u16gPvgArrowArmVoltage.AppScalingDivisor :=1;
u16gPvgArrowArmVoltage.AppScalingMultiplier :=1;
u16gPvgArrowArmVoltage.AppScalingOffset :=0;
u16gPvgArrowArmVoltage.AppUnit :="";
u16gPvgArrowArmVoltage.CanDefault :=0;
u16gPvgArrowArmVoltage.CanInit :=0;
u16gPvgArrowArmVoltage.CanMax :=VBasic.LibConst.U16_MAX;
u16gPvgArrowArmVoltage.CanMin :=VBasic.LibConst.U16_MIN;
u16gPvgArrowArmVoltage.CanUnit :="";
u16gPvgArrowArmVoltage.Description :="new signal";
u16gPvgArrowArmVoltage.ErrorReaction := eErrorReaction.ERSIG_DFLT;
u16gPvgArrowArmVoltage.ReceiverAdress :=1;
u16gPvgArrowArmVoltage.ToolScalingDivisor :=1;
u16gPvgArrowArmVoltage.ToolScalingMultiplier :=1;
u16gPvgArrowArmVoltage.ToolScalingOffset :=0;
u16gPvgArrowArmVoltage.ToolUnit :="";

u16gPvgTelescopeArmVoltage.AppScalingDivisor :=1;
u16gPvgTelescopeArmVoltage.AppScalingMultiplier :=1;
u16gPvgTelescopeArmVoltage.AppScalingOffset :=0;
u16gPvgTelescopeArmVoltage.AppUnit :="";
u16gPvgTelescopeArmVoltage.CanDefault :=0;
u16gPvgTelescopeArmVoltage.CanInit :=0;
u16gPvgTelescopeArmVoltage.CanMax :=VBasic.LibConst.U16_MAX;
u16gPvgTelescopeArmVoltage.CanMin :=VBasic.LibConst.U16_MIN;
u16gPvgTelescopeArmVoltage.CanUnit :="";
u16gPvgTelescopeArmVoltage.Description :="new signal";
u16gPvgTelescopeArmVoltage.ErrorReaction := eErrorReaction.ERSIG_DFLT;
u16gPvgTelescopeArmVoltage.ReceiverAdress :=1;
u16gPvgTelescopeArmVoltage.ToolScalingDivisor :=1;
u16gPvgTelescopeArmVoltage.ToolScalingMultiplier :=1;
u16gPvgTelescopeArmVoltage.ToolScalingOffset :=0;
u16gPvgTelescopeArmVoltage.ToolUnit :="";

u16gPvgEvTorVoltage.AppScalingDivisor :=1;
u16gPvgEvTorVoltage.AppScalingMultiplier :=1;
u16gPvgEvTorVoltage.AppScalingOffset :=0;
u16gPvgEvTorVoltage.AppUnit :="";
u16gPvgEvTorVoltage.CanDefault :=0;
u16gPvgEvTorVoltage.CanInit :=0;
u16gPvgEvTorVoltage.CanMax :=VBasic.LibConst.U16_MAX;
u16gPvgEvTorVoltage.CanMin :=VBasic.LibConst.U16_MIN;
u16gPvgEvTorVoltage.CanUnit :="";
u16gPvgEvTorVoltage.Description :="new signal";
u16gPvgEvTorVoltage.ErrorReaction := eErrorReaction.ERSIG_DFLT;
u16gPvgEvTorVoltage.ReceiverAdress :=1;
u16gPvgEvTorVoltage.ToolScalingDivisor :=1;
u16gPvgEvTorVoltage.ToolScalingMultiplier :=1;
u16gPvgEvTorVoltage.ToolScalingOffset :=0;
u16gPvgEvTorVoltage.ToolUnit :="";


                
END_METHOD
END_FUNCTION_BLOCK

FUNCTION_BLOCK Msg9C1SendToEvision7MessageClass EXTENDS CanReceiveMessageClass
  VAR_INPUT
    bogPendularMoveUp : BoolCanSignalClass;
    bogPendularMoveDown : BoolCanSignalClass;
    bogBasketRotCtClockWiseMove : BoolCanSignalClass;
    bogBasketRtClockWiseMove : BoolCanSignalClass;
    bogBasketInclinaisonMoveUp : BoolCanSignalClass;
    bogBasketInclinaisonMoveDown : BoolCanSignalClass;
    bogFuelLow : BoolCanSignalClass;
    i16gDeltaArmAngleValue : Int16CanSignalClass;
    i16gArrowArmAngleValue : Int16CanSignalClass;
    i16gTelescopePositionValue : Int16CanSignalClass;
    Counter : UInt32CanSignalClass;
  END_VAR

            
          

METHOD SetData
  VAR_INPUT
    CanMsgPointer : POINTER TO CanMessageClass;
  END_VAR
                  IF IsValidPointer(canMsgPointer,'SetData') THEN
	SUPER^.SetData(CanMsgPointer);
	//Set the new data
	bogPendularMoveUp.Value := canMsgPointer^.GetBoolOnBit(0);
	bogPendularMoveDown.Value := canMsgPointer^.GetBoolOnBit(1);
	bogBasketRotCtClockWiseMove.Value := canMsgPointer^.GetBoolOnBit(2);
	bogBasketRtClockWiseMove.Value := canMsgPointer^.GetBoolOnBit(3);
	bogBasketInclinaisonMoveUp.Value := canMsgPointer^.GetBoolOnBit(4);
	bogBasketInclinaisonMoveDown.Value := canMsgPointer^.GetBoolOnBit(5);
	bogFuelLow.Value := canMsgPointer^.GetBoolOnBit(6);
	i16gDeltaArmAngleValue.Value := canMsgPointer^.GetInt16(16);
	i16gArrowArmAngleValue.Value := canMsgPointer^.GetInt16(32);
	i16gTelescopePositionValue.Value := canMsgPointer^.GetInt16(48);
	//And increase the counter
	Counter.Value := CanMsgPointer^.Counter.Value;
END_IF

                
END_METHOD

PROPERTY bogPendularMoveUpRawValue : BOOL
GET
                    bogPendularMoveUpRawValue := bogPendularMoveUp.Value;

                  
END_GET
END_PROPERTY

PROPERTY bogPendularMoveDownRawValue : BOOL
GET
                    bogPendularMoveDownRawValue := bogPendularMoveDown.Value;

                  
END_GET
END_PROPERTY

PROPERTY bogBasketRotCtClockWiseMoveRawValue : BOOL
GET
                    bogBasketRotCtClockWiseMoveRawValue := bogBasketRotCtClockWiseMove.Value;

                  
END_GET
END_PROPERTY

PROPERTY bogBasketRtClockWiseMoveRawValue : BOOL
GET
                    bogBasketRtClockWiseMoveRawValue := bogBasketRtClockWiseMove.Value;

                  
END_GET
END_PROPERTY

PROPERTY bogBasketInclinaisonMoveUpRawValue : BOOL
GET
                    bogBasketInclinaisonMoveUpRawValue := bogBasketInclinaisonMoveUp.Value;

                  
END_GET
END_PROPERTY

PROPERTY bogBasketInclinaisonMoveDownRawValue : BOOL
GET
                    bogBasketInclinaisonMoveDownRawValue := bogBasketInclinaisonMoveDown.Value;

                  
END_GET
END_PROPERTY

PROPERTY bogFuelLowRawValue : BOOL
GET
                    bogFuelLowRawValue := bogFuelLow.Value;

                  
END_GET
END_PROPERTY

PROPERTY i16gDeltaArmAngleValueRawValue : INT
GET
                    IF i16gDeltaArmAngleValue.AppScalingMultiplier = 0 THEN
	_MatchLog^.Error("Get i16gDeltaArmAngleValueRawValue", "Division by Zero!");
	RETURN;
End_IF

i16gDeltaArmAngleValueRawValue := TO_INT((i16gDeltaArmAngleValue.Value - i16gDeltaArmAngleValue.AppScalingOffset) * i16gDeltaArmAngleValue.AppScalingDivisor / i16gDeltaArmAngleValue.AppScalingMultiplier);

                  
END_GET
END_PROPERTY

PROPERTY i16gArrowArmAngleValueRawValue : INT
GET
                    IF i16gArrowArmAngleValue.AppScalingMultiplier = 0 THEN
	_MatchLog^.Error("Get i16gArrowArmAngleValueRawValue", "Division by Zero!");
	RETURN;
End_IF

i16gArrowArmAngleValueRawValue := TO_INT((i16gArrowArmAngleValue.Value - i16gArrowArmAngleValue.AppScalingOffset) * i16gArrowArmAngleValue.AppScalingDivisor / i16gArrowArmAngleValue.AppScalingMultiplier);

                  
END_GET
END_PROPERTY

PROPERTY i16gTelescopePositionValueRawValue : INT
GET
                    IF i16gTelescopePositionValue.AppScalingMultiplier = 0 THEN
	_MatchLog^.Error("Get i16gTelescopePositionValueRawValue", "Division by Zero!");
	RETURN;
End_IF

i16gTelescopePositionValueRawValue := TO_INT((i16gTelescopePositionValue.Value - i16gTelescopePositionValue.AppScalingOffset) * i16gTelescopePositionValue.AppScalingDivisor / i16gTelescopePositionValue.AppScalingMultiplier);

                  
END_GET
END_PROPERTY

PROPERTY bogPendularMoveUpToolValue : BOOL
GET
                    bogPendularMoveUpToolValue := bogPendularMoveUp.Value;

                  
END_GET
END_PROPERTY

PROPERTY bogPendularMoveDownToolValue : BOOL
GET
                    bogPendularMoveDownToolValue := bogPendularMoveDown.Value;

                  
END_GET
END_PROPERTY

PROPERTY bogBasketRotCtClockWiseMoveToolValue : BOOL
GET
                    bogBasketRotCtClockWiseMoveToolValue := bogBasketRotCtClockWiseMove.Value;

                  
END_GET
END_PROPERTY

PROPERTY bogBasketRtClockWiseMoveToolValue : BOOL
GET
                    bogBasketRtClockWiseMoveToolValue := bogBasketRtClockWiseMove.Value;

                  
END_GET
END_PROPERTY

PROPERTY bogBasketInclinaisonMoveUpToolValue : BOOL
GET
                    bogBasketInclinaisonMoveUpToolValue := bogBasketInclinaisonMoveUp.Value;

                  
END_GET
END_PROPERTY

PROPERTY bogBasketInclinaisonMoveDownToolValue : BOOL
GET
                    bogBasketInclinaisonMoveDownToolValue := bogBasketInclinaisonMoveDown.Value;

                  
END_GET
END_PROPERTY

PROPERTY bogFuelLowToolValue : BOOL
GET
                    bogFuelLowToolValue := bogFuelLow.Value;

                  
END_GET
END_PROPERTY

PROPERTY i16gDeltaArmAngleValueToolValue : INT
GET
                    IF i16gDeltaArmAngleValue.ToolScalingDivisor = 0 OR i16gDeltaArmAngleValue.AppScalingMultiplier = 0 THEN
	_MatchLog^.Error("Get i16gDeltaArmAngleValueToolValue", "Division by Zero!");
	RETURN;
END_IF

i16gDeltaArmAngleValueToolValue := TO_INT(((i16gDeltaArmAngleValue.Value - i16gDeltaArmAngleValue.AppScalingOffset) * i16gDeltaArmAngleValue.AppScalingDivisor / i16gDeltaArmAngleValue.AppScalingMultiplier * i16gDeltaArmAngleValue.ToolScalingMultiplier / i16gDeltaArmAngleValue.ToolScalingDivisor) + i16gDeltaArmAngleValue.ToolScalingOffset);

                  
END_GET
END_PROPERTY

PROPERTY i16gArrowArmAngleValueToolValue : INT
GET
                    IF i16gArrowArmAngleValue.ToolScalingDivisor = 0 OR i16gArrowArmAngleValue.AppScalingMultiplier = 0 THEN
	_MatchLog^.Error("Get i16gArrowArmAngleValueToolValue", "Division by Zero!");
	RETURN;
END_IF

i16gArrowArmAngleValueToolValue := TO_INT(((i16gArrowArmAngleValue.Value - i16gArrowArmAngleValue.AppScalingOffset) * i16gArrowArmAngleValue.AppScalingDivisor / i16gArrowArmAngleValue.AppScalingMultiplier * i16gArrowArmAngleValue.ToolScalingMultiplier / i16gArrowArmAngleValue.ToolScalingDivisor) + i16gArrowArmAngleValue.ToolScalingOffset);

                  
END_GET
END_PROPERTY

PROPERTY i16gTelescopePositionValueToolValue : INT
GET
                    IF i16gTelescopePositionValue.ToolScalingDivisor = 0 OR i16gTelescopePositionValue.AppScalingMultiplier = 0 THEN
	_MatchLog^.Error("Get i16gTelescopePositionValueToolValue", "Division by Zero!");
	RETURN;
END_IF

i16gTelescopePositionValueToolValue := TO_INT(((i16gTelescopePositionValue.Value - i16gTelescopePositionValue.AppScalingOffset) * i16gTelescopePositionValue.AppScalingDivisor / i16gTelescopePositionValue.AppScalingMultiplier * i16gTelescopePositionValue.ToolScalingMultiplier / i16gTelescopePositionValue.ToolScalingDivisor) + i16gTelescopePositionValue.ToolScalingOffset);

                  
END_GET
END_PROPERTY

METHOD InitializeCanSignals
                  bogPendularMoveUp.AppScalingDivisor :=1;
bogPendularMoveUp.AppScalingMultiplier :=1;
bogPendularMoveUp.AppScalingOffset :=0;
bogPendularMoveUp.AppUnit :="";
bogPendularMoveUp.CanDefault :=0;
bogPendularMoveUp.CanInit :=0;
bogPendularMoveUp.CanMax :=1;
bogPendularMoveUp.CanMin :=0;
bogPendularMoveUp.CanUnit :="";
bogPendularMoveUp.Description :="new signal";
bogPendularMoveUp.ErrorReaction := eErrorReaction.ERSIG_DFLT;
bogPendularMoveUp.ReceiverAdress :=1;
bogPendularMoveUp.ToolScalingDivisor :=1;
bogPendularMoveUp.ToolScalingMultiplier :=1;
bogPendularMoveUp.ToolScalingOffset :=0;
bogPendularMoveUp.ToolUnit :="";

bogPendularMoveDown.AppScalingDivisor :=1;
bogPendularMoveDown.AppScalingMultiplier :=1;
bogPendularMoveDown.AppScalingOffset :=0;
bogPendularMoveDown.AppUnit :="";
bogPendularMoveDown.CanDefault :=0;
bogPendularMoveDown.CanInit :=0;
bogPendularMoveDown.CanMax :=1;
bogPendularMoveDown.CanMin :=0;
bogPendularMoveDown.CanUnit :="";
bogPendularMoveDown.Description :="new signal";
bogPendularMoveDown.ErrorReaction := eErrorReaction.ERSIG_DFLT;
bogPendularMoveDown.ReceiverAdress :=1;
bogPendularMoveDown.ToolScalingDivisor :=1;
bogPendularMoveDown.ToolScalingMultiplier :=1;
bogPendularMoveDown.ToolScalingOffset :=0;
bogPendularMoveDown.ToolUnit :="";

bogBasketRotCtClockWiseMove.AppScalingDivisor :=1;
bogBasketRotCtClockWiseMove.AppScalingMultiplier :=1;
bogBasketRotCtClockWiseMove.AppScalingOffset :=0;
bogBasketRotCtClockWiseMove.AppUnit :="";
bogBasketRotCtClockWiseMove.CanDefault :=0;
bogBasketRotCtClockWiseMove.CanInit :=0;
bogBasketRotCtClockWiseMove.CanMax :=1;
bogBasketRotCtClockWiseMove.CanMin :=0;
bogBasketRotCtClockWiseMove.CanUnit :="";
bogBasketRotCtClockWiseMove.Description :="new signal";
bogBasketRotCtClockWiseMove.ErrorReaction := eErrorReaction.ERSIG_DFLT;
bogBasketRotCtClockWiseMove.ReceiverAdress :=1;
bogBasketRotCtClockWiseMove.ToolScalingDivisor :=1;
bogBasketRotCtClockWiseMove.ToolScalingMultiplier :=1;
bogBasketRotCtClockWiseMove.ToolScalingOffset :=0;
bogBasketRotCtClockWiseMove.ToolUnit :="";

bogBasketRtClockWiseMove.AppScalingDivisor :=1;
bogBasketRtClockWiseMove.AppScalingMultiplier :=1;
bogBasketRtClockWiseMove.AppScalingOffset :=0;
bogBasketRtClockWiseMove.AppUnit :="";
bogBasketRtClockWiseMove.CanDefault :=0;
bogBasketRtClockWiseMove.CanInit :=0;
bogBasketRtClockWiseMove.CanMax :=1;
bogBasketRtClockWiseMove.CanMin :=0;
bogBasketRtClockWiseMove.CanUnit :="";
bogBasketRtClockWiseMove.Description :="new signal";
bogBasketRtClockWiseMove.ErrorReaction := eErrorReaction.ERSIG_DFLT;
bogBasketRtClockWiseMove.ReceiverAdress :=1;
bogBasketRtClockWiseMove.ToolScalingDivisor :=1;
bogBasketRtClockWiseMove.ToolScalingMultiplier :=1;
bogBasketRtClockWiseMove.ToolScalingOffset :=0;
bogBasketRtClockWiseMove.ToolUnit :="";

bogBasketInclinaisonMoveUp.AppScalingDivisor :=1;
bogBasketInclinaisonMoveUp.AppScalingMultiplier :=1;
bogBasketInclinaisonMoveUp.AppScalingOffset :=0;
bogBasketInclinaisonMoveUp.AppUnit :="";
bogBasketInclinaisonMoveUp.CanDefault :=0;
bogBasketInclinaisonMoveUp.CanInit :=0;
bogBasketInclinaisonMoveUp.CanMax :=1;
bogBasketInclinaisonMoveUp.CanMin :=0;
bogBasketInclinaisonMoveUp.CanUnit :="";
bogBasketInclinaisonMoveUp.Description :="new signal";
bogBasketInclinaisonMoveUp.ErrorReaction := eErrorReaction.ERSIG_DFLT;
bogBasketInclinaisonMoveUp.ReceiverAdress :=1;
bogBasketInclinaisonMoveUp.ToolScalingDivisor :=1;
bogBasketInclinaisonMoveUp.ToolScalingMultiplier :=1;
bogBasketInclinaisonMoveUp.ToolScalingOffset :=0;
bogBasketInclinaisonMoveUp.ToolUnit :="";

bogBasketInclinaisonMoveDown.AppScalingDivisor :=1;
bogBasketInclinaisonMoveDown.AppScalingMultiplier :=1;
bogBasketInclinaisonMoveDown.AppScalingOffset :=0;
bogBasketInclinaisonMoveDown.AppUnit :="";
bogBasketInclinaisonMoveDown.CanDefault :=0;
bogBasketInclinaisonMoveDown.CanInit :=0;
bogBasketInclinaisonMoveDown.CanMax :=1;
bogBasketInclinaisonMoveDown.CanMin :=0;
bogBasketInclinaisonMoveDown.CanUnit :="";
bogBasketInclinaisonMoveDown.Description :="new signal";
bogBasketInclinaisonMoveDown.ErrorReaction := eErrorReaction.ERSIG_DFLT;
bogBasketInclinaisonMoveDown.ReceiverAdress :=1;
bogBasketInclinaisonMoveDown.ToolScalingDivisor :=1;
bogBasketInclinaisonMoveDown.ToolScalingMultiplier :=1;
bogBasketInclinaisonMoveDown.ToolScalingOffset :=0;
bogBasketInclinaisonMoveDown.ToolUnit :="";

bogFuelLow.AppScalingDivisor :=1;
bogFuelLow.AppScalingMultiplier :=1;
bogFuelLow.AppScalingOffset :=0;
bogFuelLow.AppUnit :="";
bogFuelLow.CanDefault :=0;
bogFuelLow.CanInit :=0;
bogFuelLow.CanMax :=1;
bogFuelLow.CanMin :=0;
bogFuelLow.CanUnit :="";
bogFuelLow.Description :="new signal";
bogFuelLow.ErrorReaction := eErrorReaction.ERSIG_DFLT;
bogFuelLow.ReceiverAdress :=1;
bogFuelLow.ToolScalingDivisor :=1;
bogFuelLow.ToolScalingMultiplier :=1;
bogFuelLow.ToolScalingOffset :=0;
bogFuelLow.ToolUnit :="";

i16gDeltaArmAngleValue.AppScalingDivisor :=1;
i16gDeltaArmAngleValue.AppScalingMultiplier :=1;
i16gDeltaArmAngleValue.AppScalingOffset :=0;
i16gDeltaArmAngleValue.AppUnit :="";
i16gDeltaArmAngleValue.CanDefault :=0;
i16gDeltaArmAngleValue.CanInit :=0;
i16gDeltaArmAngleValue.CanMax :=VBasic.LibConst.I16_MAX;
i16gDeltaArmAngleValue.CanMin :=VBasic.LibConst.I16_MIN;
i16gDeltaArmAngleValue.CanUnit :="";
i16gDeltaArmAngleValue.Description :="new signal";
i16gDeltaArmAngleValue.ErrorReaction := eErrorReaction.ERSIG_DFLT;
i16gDeltaArmAngleValue.ReceiverAdress :=1;
i16gDeltaArmAngleValue.ToolScalingDivisor :=1;
i16gDeltaArmAngleValue.ToolScalingMultiplier :=1;
i16gDeltaArmAngleValue.ToolScalingOffset :=0;
i16gDeltaArmAngleValue.ToolUnit :="";

i16gArrowArmAngleValue.AppScalingDivisor :=1;
i16gArrowArmAngleValue.AppScalingMultiplier :=1;
i16gArrowArmAngleValue.AppScalingOffset :=0;
i16gArrowArmAngleValue.AppUnit :="";
i16gArrowArmAngleValue.CanDefault :=0;
i16gArrowArmAngleValue.CanInit :=0;
i16gArrowArmAngleValue.CanMax :=VBasic.LibConst.I16_MAX;
i16gArrowArmAngleValue.CanMin :=VBasic.LibConst.I16_MIN;
i16gArrowArmAngleValue.CanUnit :="";
i16gArrowArmAngleValue.Description :="new signal";
i16gArrowArmAngleValue.ErrorReaction := eErrorReaction.ERSIG_DFLT;
i16gArrowArmAngleValue.ReceiverAdress :=1;
i16gArrowArmAngleValue.ToolScalingDivisor :=1;
i16gArrowArmAngleValue.ToolScalingMultiplier :=1;
i16gArrowArmAngleValue.ToolScalingOffset :=0;
i16gArrowArmAngleValue.ToolUnit :="";

i16gTelescopePositionValue.AppScalingDivisor :=1;
i16gTelescopePositionValue.AppScalingMultiplier :=1;
i16gTelescopePositionValue.AppScalingOffset :=0;
i16gTelescopePositionValue.AppUnit :="";
i16gTelescopePositionValue.CanDefault :=0;
i16gTelescopePositionValue.CanInit :=0;
i16gTelescopePositionValue.CanMax :=VBasic.LibConst.I16_MAX;
i16gTelescopePositionValue.CanMin :=VBasic.LibConst.I16_MIN;
i16gTelescopePositionValue.CanUnit :="";
i16gTelescopePositionValue.Description :="new signal";
i16gTelescopePositionValue.ErrorReaction := eErrorReaction.ERSIG_DFLT;
i16gTelescopePositionValue.ReceiverAdress :=1;
i16gTelescopePositionValue.ToolScalingDivisor :=1;
i16gTelescopePositionValue.ToolScalingMultiplier :=1;
i16gTelescopePositionValue.ToolScalingOffset :=0;
i16gTelescopePositionValue.ToolUnit :="";


                
END_METHOD
END_FUNCTION_BLOCK

FUNCTION_BLOCK Msg10C1SendToEvision7MessageClass EXTENDS CanReceiveMessageClass
  VAR_INPUT
    u8gTTC510Version_Major : UInt8CanSignalClass;
    u8gTTC510Version_Minor : UInt8CanSignalClass;
    u8gTTC510Version_Patch : UInt8CanSignalClass;
    u8gTTC510Version_Custom : UInt8CanSignalClass;
    u8gTTC48XSVersion_Major : UInt8CanSignalClass;
    u8gTTC48XSVersion_Minor : UInt8CanSignalClass;
    u8gTTC48XSVersion_Patch : UInt8CanSignalClass;
    u8gTTC48XSVersion_Custom : UInt8CanSignalClass;
    Counter : UInt32CanSignalClass;
  END_VAR

            
          

METHOD SetData
  VAR_INPUT
    CanMsgPointer : POINTER TO CanMessageClass;
  END_VAR
                  IF IsValidPointer(canMsgPointer,'SetData') THEN
	SUPER^.SetData(CanMsgPointer);
	//Set the new data
	u8gTTC510Version_Major.Value := canMsgPointer^.GetUint8(0);
	u8gTTC510Version_Minor.Value := canMsgPointer^.GetUint8(8);
	u8gTTC510Version_Patch.Value := canMsgPointer^.GetUint8(16);
	u8gTTC510Version_Custom.Value := canMsgPointer^.GetUint8(24);
	u8gTTC48XSVersion_Major.Value := canMsgPointer^.GetUint8(32);
	u8gTTC48XSVersion_Minor.Value := canMsgPointer^.GetUint8(40);
	u8gTTC48XSVersion_Patch.Value := canMsgPointer^.GetUint8(48);
	u8gTTC48XSVersion_Custom.Value := canMsgPointer^.GetUint8(56);
	//And increase the counter
	Counter.Value := CanMsgPointer^.Counter.Value;
END_IF

                
END_METHOD

PROPERTY u8gTTC510Version_MajorRawValue : USINT
GET
                    IF u8gTTC510Version_Major.AppScalingMultiplier = 0 THEN
	_MatchLog^.Error("Get u8gTTC510Version_MajorRawValue", "Division by Zero!");
	RETURN;
End_IF

u8gTTC510Version_MajorRawValue := TO_USINT((u8gTTC510Version_Major.Value - u8gTTC510Version_Major.AppScalingOffset) * u8gTTC510Version_Major.AppScalingDivisor / u8gTTC510Version_Major.AppScalingMultiplier);

                  
END_GET
END_PROPERTY

PROPERTY u8gTTC510Version_MinorRawValue : USINT
GET
                    IF u8gTTC510Version_Minor.AppScalingMultiplier = 0 THEN
	_MatchLog^.Error("Get u8gTTC510Version_MinorRawValue", "Division by Zero!");
	RETURN;
End_IF

u8gTTC510Version_MinorRawValue := TO_USINT((u8gTTC510Version_Minor.Value - u8gTTC510Version_Minor.AppScalingOffset) * u8gTTC510Version_Minor.AppScalingDivisor / u8gTTC510Version_Minor.AppScalingMultiplier);

                  
END_GET
END_PROPERTY

PROPERTY u8gTTC510Version_PatchRawValue : USINT
GET
                    IF u8gTTC510Version_Patch.AppScalingMultiplier = 0 THEN
	_MatchLog^.Error("Get u8gTTC510Version_PatchRawValue", "Division by Zero!");
	RETURN;
End_IF

u8gTTC510Version_PatchRawValue := TO_USINT((u8gTTC510Version_Patch.Value - u8gTTC510Version_Patch.AppScalingOffset) * u8gTTC510Version_Patch.AppScalingDivisor / u8gTTC510Version_Patch.AppScalingMultiplier);

                  
END_GET
END_PROPERTY

PROPERTY u8gTTC510Version_CustomRawValue : USINT
GET
                    IF u8gTTC510Version_Custom.AppScalingMultiplier = 0 THEN
	_MatchLog^.Error("Get u8gTTC510Version_CustomRawValue", "Division by Zero!");
	RETURN;
End_IF

u8gTTC510Version_CustomRawValue := TO_USINT((u8gTTC510Version_Custom.Value - u8gTTC510Version_Custom.AppScalingOffset) * u8gTTC510Version_Custom.AppScalingDivisor / u8gTTC510Version_Custom.AppScalingMultiplier);

                  
END_GET
END_PROPERTY

PROPERTY u8gTTC48XSVersion_MajorRawValue : USINT
GET
                    IF u8gTTC48XSVersion_Major.AppScalingMultiplier = 0 THEN
	_MatchLog^.Error("Get u8gTTC48XSVersion_MajorRawValue", "Division by Zero!");
	RETURN;
End_IF

u8gTTC48XSVersion_MajorRawValue := TO_USINT((u8gTTC48XSVersion_Major.Value - u8gTTC48XSVersion_Major.AppScalingOffset) * u8gTTC48XSVersion_Major.AppScalingDivisor / u8gTTC48XSVersion_Major.AppScalingMultiplier);

                  
END_GET
END_PROPERTY

PROPERTY u8gTTC48XSVersion_MinorRawValue : USINT
GET
                    IF u8gTTC48XSVersion_Minor.AppScalingMultiplier = 0 THEN
	_MatchLog^.Error("Get u8gTTC48XSVersion_MinorRawValue", "Division by Zero!");
	RETURN;
End_IF

u8gTTC48XSVersion_MinorRawValue := TO_USINT((u8gTTC48XSVersion_Minor.Value - u8gTTC48XSVersion_Minor.AppScalingOffset) * u8gTTC48XSVersion_Minor.AppScalingDivisor / u8gTTC48XSVersion_Minor.AppScalingMultiplier);

                  
END_GET
END_PROPERTY

PROPERTY u8gTTC48XSVersion_PatchRawValue : USINT
GET
                    IF u8gTTC48XSVersion_Patch.AppScalingMultiplier = 0 THEN
	_MatchLog^.Error("Get u8gTTC48XSVersion_PatchRawValue", "Division by Zero!");
	RETURN;
End_IF

u8gTTC48XSVersion_PatchRawValue := TO_USINT((u8gTTC48XSVersion_Patch.Value - u8gTTC48XSVersion_Patch.AppScalingOffset) * u8gTTC48XSVersion_Patch.AppScalingDivisor / u8gTTC48XSVersion_Patch.AppScalingMultiplier);

                  
END_GET
END_PROPERTY

PROPERTY u8gTTC48XSVersion_CustomRawValue : USINT
GET
                    IF u8gTTC48XSVersion_Custom.AppScalingMultiplier = 0 THEN
	_MatchLog^.Error("Get u8gTTC48XSVersion_CustomRawValue", "Division by Zero!");
	RETURN;
End_IF

u8gTTC48XSVersion_CustomRawValue := TO_USINT((u8gTTC48XSVersion_Custom.Value - u8gTTC48XSVersion_Custom.AppScalingOffset) * u8gTTC48XSVersion_Custom.AppScalingDivisor / u8gTTC48XSVersion_Custom.AppScalingMultiplier);

                  
END_GET
END_PROPERTY

PROPERTY u8gTTC510Version_MajorToolValue : USINT
GET
                    IF u8gTTC510Version_Major.ToolScalingDivisor = 0 OR u8gTTC510Version_Major.AppScalingMultiplier = 0 THEN
	_MatchLog^.Error("Get u8gTTC510Version_MajorToolValue", "Division by Zero!");
	RETURN;
END_IF

u8gTTC510Version_MajorToolValue := TO_USINT(((u8gTTC510Version_Major.Value - u8gTTC510Version_Major.AppScalingOffset) * u8gTTC510Version_Major.AppScalingDivisor / u8gTTC510Version_Major.AppScalingMultiplier * u8gTTC510Version_Major.ToolScalingMultiplier / u8gTTC510Version_Major.ToolScalingDivisor) + u8gTTC510Version_Major.ToolScalingOffset);

                  
END_GET
END_PROPERTY

PROPERTY u8gTTC510Version_MinorToolValue : USINT
GET
                    IF u8gTTC510Version_Minor.ToolScalingDivisor = 0 OR u8gTTC510Version_Minor.AppScalingMultiplier = 0 THEN
	_MatchLog^.Error("Get u8gTTC510Version_MinorToolValue", "Division by Zero!");
	RETURN;
END_IF

u8gTTC510Version_MinorToolValue := TO_USINT(((u8gTTC510Version_Minor.Value - u8gTTC510Version_Minor.AppScalingOffset) * u8gTTC510Version_Minor.AppScalingDivisor / u8gTTC510Version_Minor.AppScalingMultiplier * u8gTTC510Version_Minor.ToolScalingMultiplier / u8gTTC510Version_Minor.ToolScalingDivisor) + u8gTTC510Version_Minor.ToolScalingOffset);

                  
END_GET
END_PROPERTY

PROPERTY u8gTTC510Version_PatchToolValue : USINT
GET
                    IF u8gTTC510Version_Patch.ToolScalingDivisor = 0 OR u8gTTC510Version_Patch.AppScalingMultiplier = 0 THEN
	_MatchLog^.Error("Get u8gTTC510Version_PatchToolValue", "Division by Zero!");
	RETURN;
END_IF

u8gTTC510Version_PatchToolValue := TO_USINT(((u8gTTC510Version_Patch.Value - u8gTTC510Version_Patch.AppScalingOffset) * u8gTTC510Version_Patch.AppScalingDivisor / u8gTTC510Version_Patch.AppScalingMultiplier * u8gTTC510Version_Patch.ToolScalingMultiplier / u8gTTC510Version_Patch.ToolScalingDivisor) + u8gTTC510Version_Patch.ToolScalingOffset);

                  
END_GET
END_PROPERTY

PROPERTY u8gTTC510Version_CustomToolValue : USINT
GET
                    IF u8gTTC510Version_Custom.ToolScalingDivisor = 0 OR u8gTTC510Version_Custom.AppScalingMultiplier = 0 THEN
	_MatchLog^.Error("Get u8gTTC510Version_CustomToolValue", "Division by Zero!");
	RETURN;
END_IF

u8gTTC510Version_CustomToolValue := TO_USINT(((u8gTTC510Version_Custom.Value - u8gTTC510Version_Custom.AppScalingOffset) * u8gTTC510Version_Custom.AppScalingDivisor / u8gTTC510Version_Custom.AppScalingMultiplier * u8gTTC510Version_Custom.ToolScalingMultiplier / u8gTTC510Version_Custom.ToolScalingDivisor) + u8gTTC510Version_Custom.ToolScalingOffset);

                  
END_GET
END_PROPERTY

PROPERTY u8gTTC48XSVersion_MajorToolValue : USINT
GET
                    IF u8gTTC48XSVersion_Major.ToolScalingDivisor = 0 OR u8gTTC48XSVersion_Major.AppScalingMultiplier = 0 THEN
	_MatchLog^.Error("Get u8gTTC48XSVersion_MajorToolValue", "Division by Zero!");
	RETURN;
END_IF

u8gTTC48XSVersion_MajorToolValue := TO_USINT(((u8gTTC48XSVersion_Major.Value - u8gTTC48XSVersion_Major.AppScalingOffset) * u8gTTC48XSVersion_Major.AppScalingDivisor / u8gTTC48XSVersion_Major.AppScalingMultiplier * u8gTTC48XSVersion_Major.ToolScalingMultiplier / u8gTTC48XSVersion_Major.ToolScalingDivisor) + u8gTTC48XSVersion_Major.ToolScalingOffset);

                  
END_GET
END_PROPERTY

PROPERTY u8gTTC48XSVersion_MinorToolValue : USINT
GET
                    IF u8gTTC48XSVersion_Minor.ToolScalingDivisor = 0 OR u8gTTC48XSVersion_Minor.AppScalingMultiplier = 0 THEN
	_MatchLog^.Error("Get u8gTTC48XSVersion_MinorToolValue", "Division by Zero!");
	RETURN;
END_IF

u8gTTC48XSVersion_MinorToolValue := TO_USINT(((u8gTTC48XSVersion_Minor.Value - u8gTTC48XSVersion_Minor.AppScalingOffset) * u8gTTC48XSVersion_Minor.AppScalingDivisor / u8gTTC48XSVersion_Minor.AppScalingMultiplier * u8gTTC48XSVersion_Minor.ToolScalingMultiplier / u8gTTC48XSVersion_Minor.ToolScalingDivisor) + u8gTTC48XSVersion_Minor.ToolScalingOffset);

                  
END_GET
END_PROPERTY

PROPERTY u8gTTC48XSVersion_PatchToolValue : USINT
GET
                    IF u8gTTC48XSVersion_Patch.ToolScalingDivisor = 0 OR u8gTTC48XSVersion_Patch.AppScalingMultiplier = 0 THEN
	_MatchLog^.Error("Get u8gTTC48XSVersion_PatchToolValue", "Division by Zero!");
	RETURN;
END_IF

u8gTTC48XSVersion_PatchToolValue := TO_USINT(((u8gTTC48XSVersion_Patch.Value - u8gTTC48XSVersion_Patch.AppScalingOffset) * u8gTTC48XSVersion_Patch.AppScalingDivisor / u8gTTC48XSVersion_Patch.AppScalingMultiplier * u8gTTC48XSVersion_Patch.ToolScalingMultiplier / u8gTTC48XSVersion_Patch.ToolScalingDivisor) + u8gTTC48XSVersion_Patch.ToolScalingOffset);

                  
END_GET
END_PROPERTY

PROPERTY u8gTTC48XSVersion_CustomToolValue : USINT
GET
                    IF u8gTTC48XSVersion_Custom.ToolScalingDivisor = 0 OR u8gTTC48XSVersion_Custom.AppScalingMultiplier = 0 THEN
	_MatchLog^.Error("Get u8gTTC48XSVersion_CustomToolValue", "Division by Zero!");
	RETURN;
END_IF

u8gTTC48XSVersion_CustomToolValue := TO_USINT(((u8gTTC48XSVersion_Custom.Value - u8gTTC48XSVersion_Custom.AppScalingOffset) * u8gTTC48XSVersion_Custom.AppScalingDivisor / u8gTTC48XSVersion_Custom.AppScalingMultiplier * u8gTTC48XSVersion_Custom.ToolScalingMultiplier / u8gTTC48XSVersion_Custom.ToolScalingDivisor) + u8gTTC48XSVersion_Custom.ToolScalingOffset);

                  
END_GET
END_PROPERTY

METHOD InitializeCanSignals
                  u8gTTC510Version_Major.AppScalingDivisor :=1;
u8gTTC510Version_Major.AppScalingMultiplier :=1;
u8gTTC510Version_Major.AppScalingOffset :=0;
u8gTTC510Version_Major.AppUnit :="";
u8gTTC510Version_Major.CanDefault :=0;
u8gTTC510Version_Major.CanInit :=0;
u8gTTC510Version_Major.CanMax :=VBasic.LibConst.U8_MAX;
u8gTTC510Version_Major.CanMin :=VBasic.LibConst.U8_MIN;
u8gTTC510Version_Major.CanUnit :="";
u8gTTC510Version_Major.Description :="Program Version Major C1 TTC510";
u8gTTC510Version_Major.ErrorReaction := eErrorReaction.ERSIG_DFLT;
u8gTTC510Version_Major.ReceiverAdress :=1;
u8gTTC510Version_Major.ToolScalingDivisor :=1;
u8gTTC510Version_Major.ToolScalingMultiplier :=1;
u8gTTC510Version_Major.ToolScalingOffset :=0;
u8gTTC510Version_Major.ToolUnit :="";

u8gTTC510Version_Minor.AppScalingDivisor :=1;
u8gTTC510Version_Minor.AppScalingMultiplier :=1;
u8gTTC510Version_Minor.AppScalingOffset :=0;
u8gTTC510Version_Minor.AppUnit :="";
u8gTTC510Version_Minor.CanDefault :=0;
u8gTTC510Version_Minor.CanInit :=0;
u8gTTC510Version_Minor.CanMax :=VBasic.LibConst.U8_MAX;
u8gTTC510Version_Minor.CanMin :=VBasic.LibConst.U8_MIN;
u8gTTC510Version_Minor.CanUnit :="";
u8gTTC510Version_Minor.Description :="Program Version Minor C1 TTC510";
u8gTTC510Version_Minor.ErrorReaction := eErrorReaction.ERSIG_DFLT;
u8gTTC510Version_Minor.ReceiverAdress :=1;
u8gTTC510Version_Minor.ToolScalingDivisor :=1;
u8gTTC510Version_Minor.ToolScalingMultiplier :=1;
u8gTTC510Version_Minor.ToolScalingOffset :=0;
u8gTTC510Version_Minor.ToolUnit :="";

u8gTTC510Version_Patch.AppScalingDivisor :=1;
u8gTTC510Version_Patch.AppScalingMultiplier :=1;
u8gTTC510Version_Patch.AppScalingOffset :=0;
u8gTTC510Version_Patch.AppUnit :="";
u8gTTC510Version_Patch.CanDefault :=0;
u8gTTC510Version_Patch.CanInit :=0;
u8gTTC510Version_Patch.CanMax :=VBasic.LibConst.U8_MAX;
u8gTTC510Version_Patch.CanMin :=VBasic.LibConst.U8_MIN;
u8gTTC510Version_Patch.CanUnit :="";
u8gTTC510Version_Patch.Description :="Program Version Patch C1 TTC510";
u8gTTC510Version_Patch.ErrorReaction := eErrorReaction.ERSIG_DFLT;
u8gTTC510Version_Patch.ReceiverAdress :=1;
u8gTTC510Version_Patch.ToolScalingDivisor :=1;
u8gTTC510Version_Patch.ToolScalingMultiplier :=1;
u8gTTC510Version_Patch.ToolScalingOffset :=0;
u8gTTC510Version_Patch.ToolUnit :="";

u8gTTC510Version_Custom.AppScalingDivisor :=1;
u8gTTC510Version_Custom.AppScalingMultiplier :=1;
u8gTTC510Version_Custom.AppScalingOffset :=0;
u8gTTC510Version_Custom.AppUnit :="";
u8gTTC510Version_Custom.CanDefault :=0;
u8gTTC510Version_Custom.CanInit :=0;
u8gTTC510Version_Custom.CanMax :=VBasic.LibConst.U8_MAX;
u8gTTC510Version_Custom.CanMin :=VBasic.LibConst.U8_MIN;
u8gTTC510Version_Custom.CanUnit :="";
u8gTTC510Version_Custom.Description :="Program Version Custom C1 TTC510";
u8gTTC510Version_Custom.ErrorReaction := eErrorReaction.ERSIG_DFLT;
u8gTTC510Version_Custom.ReceiverAdress :=1;
u8gTTC510Version_Custom.ToolScalingDivisor :=1;
u8gTTC510Version_Custom.ToolScalingMultiplier :=1;
u8gTTC510Version_Custom.ToolScalingOffset :=0;
u8gTTC510Version_Custom.ToolUnit :="";

u8gTTC48XSVersion_Major.AppScalingDivisor :=1;
u8gTTC48XSVersion_Major.AppScalingMultiplier :=1;
u8gTTC48XSVersion_Major.AppScalingOffset :=0;
u8gTTC48XSVersion_Major.AppUnit :="";
u8gTTC48XSVersion_Major.CanDefault :=0;
u8gTTC48XSVersion_Major.CanInit :=0;
u8gTTC48XSVersion_Major.CanMax :=VBasic.LibConst.U8_MAX;
u8gTTC48XSVersion_Major.CanMin :=VBasic.LibConst.U8_MIN;
u8gTTC48XSVersion_Major.CanUnit :="";
u8gTTC48XSVersion_Major.Description :="Program Version Major TTC48XS";
u8gTTC48XSVersion_Major.ErrorReaction := eErrorReaction.ERSIG_DFLT;
u8gTTC48XSVersion_Major.ReceiverAdress :=1;
u8gTTC48XSVersion_Major.ToolScalingDivisor :=1;
u8gTTC48XSVersion_Major.ToolScalingMultiplier :=1;
u8gTTC48XSVersion_Major.ToolScalingOffset :=0;
u8gTTC48XSVersion_Major.ToolUnit :="";

u8gTTC48XSVersion_Minor.AppScalingDivisor :=1;
u8gTTC48XSVersion_Minor.AppScalingMultiplier :=1;
u8gTTC48XSVersion_Minor.AppScalingOffset :=0;
u8gTTC48XSVersion_Minor.AppUnit :="";
u8gTTC48XSVersion_Minor.CanDefault :=0;
u8gTTC48XSVersion_Minor.CanInit :=0;
u8gTTC48XSVersion_Minor.CanMax :=VBasic.LibConst.U8_MAX;
u8gTTC48XSVersion_Minor.CanMin :=VBasic.LibConst.U8_MIN;
u8gTTC48XSVersion_Minor.CanUnit :="";
u8gTTC48XSVersion_Minor.Description :="Program Version MinorTTC48XS";
u8gTTC48XSVersion_Minor.ErrorReaction := eErrorReaction.ERSIG_DFLT;
u8gTTC48XSVersion_Minor.ReceiverAdress :=1;
u8gTTC48XSVersion_Minor.ToolScalingDivisor :=1;
u8gTTC48XSVersion_Minor.ToolScalingMultiplier :=1;
u8gTTC48XSVersion_Minor.ToolScalingOffset :=0;
u8gTTC48XSVersion_Minor.ToolUnit :="";

u8gTTC48XSVersion_Patch.AppScalingDivisor :=1;
u8gTTC48XSVersion_Patch.AppScalingMultiplier :=1;
u8gTTC48XSVersion_Patch.AppScalingOffset :=0;
u8gTTC48XSVersion_Patch.AppUnit :="";
u8gTTC48XSVersion_Patch.CanDefault :=0;
u8gTTC48XSVersion_Patch.CanInit :=0;
u8gTTC48XSVersion_Patch.CanMax :=VBasic.LibConst.U8_MAX;
u8gTTC48XSVersion_Patch.CanMin :=VBasic.LibConst.U8_MIN;
u8gTTC48XSVersion_Patch.CanUnit :="";
u8gTTC48XSVersion_Patch.Description :="Program Version Patch TTC48XS";
u8gTTC48XSVersion_Patch.ErrorReaction := eErrorReaction.ERSIG_DFLT;
u8gTTC48XSVersion_Patch.ReceiverAdress :=1;
u8gTTC48XSVersion_Patch.ToolScalingDivisor :=1;
u8gTTC48XSVersion_Patch.ToolScalingMultiplier :=1;
u8gTTC48XSVersion_Patch.ToolScalingOffset :=0;
u8gTTC48XSVersion_Patch.ToolUnit :="";

u8gTTC48XSVersion_Custom.AppScalingDivisor :=1;
u8gTTC48XSVersion_Custom.AppScalingMultiplier :=1;
u8gTTC48XSVersion_Custom.AppScalingOffset :=0;
u8gTTC48XSVersion_Custom.AppUnit :="";
u8gTTC48XSVersion_Custom.CanDefault :=0;
u8gTTC48XSVersion_Custom.CanInit :=0;
u8gTTC48XSVersion_Custom.CanMax :=VBasic.LibConst.U8_MAX;
u8gTTC48XSVersion_Custom.CanMin :=VBasic.LibConst.U8_MIN;
u8gTTC48XSVersion_Custom.CanUnit :="";
u8gTTC48XSVersion_Custom.Description :="Program Version Custom TTC48XS";
u8gTTC48XSVersion_Custom.ErrorReaction := eErrorReaction.ERSIG_DFLT;
u8gTTC48XSVersion_Custom.ReceiverAdress :=1;
u8gTTC48XSVersion_Custom.ToolScalingDivisor :=1;
u8gTTC48XSVersion_Custom.ToolScalingMultiplier :=1;
u8gTTC48XSVersion_Custom.ToolScalingOffset :=0;
u8gTTC48XSVersion_Custom.ToolUnit :="";


                
END_METHOD
END_FUNCTION_BLOCK

FUNCTION_BLOCK Msg11C1SendToEvision7MessageClass EXTENDS CanReceiveMessageClass
  VAR_INPUT
    i16gScalingJoysTurret : Int16CanSignalClass;
    i16gScalingJoysDeltaArm : Int16CanSignalClass;
    i16gScalingJoysArrowArm : Int16CanSignalClass;
    i16gScalingJoysTelescopeArm : Int16CanSignalClass;
    Counter : UInt32CanSignalClass;
  END_VAR

            
          

METHOD SetData
  VAR_INPUT
    CanMsgPointer : POINTER TO CanMessageClass;
  END_VAR
                  IF IsValidPointer(canMsgPointer,'SetData') THEN
	SUPER^.SetData(CanMsgPointer);
	//Set the new data
	i16gScalingJoysTurret.Value := canMsgPointer^.GetInt16(0);
	i16gScalingJoysDeltaArm.Value := canMsgPointer^.GetInt16(16);
	i16gScalingJoysArrowArm.Value := canMsgPointer^.GetInt16(32);
	i16gScalingJoysTelescopeArm.Value := canMsgPointer^.GetInt16(48);
	//And increase the counter
	Counter.Value := CanMsgPointer^.Counter.Value;
END_IF

                
END_METHOD

PROPERTY i16gScalingJoysTurretRawValue : INT
GET
                    IF i16gScalingJoysTurret.AppScalingMultiplier = 0 THEN
	_MatchLog^.Error("Get i16gScalingJoysTurretRawValue", "Division by Zero!");
	RETURN;
End_IF

i16gScalingJoysTurretRawValue := TO_INT((i16gScalingJoysTurret.Value - i16gScalingJoysTurret.AppScalingOffset) * i16gScalingJoysTurret.AppScalingDivisor / i16gScalingJoysTurret.AppScalingMultiplier);

                  
END_GET
END_PROPERTY

PROPERTY i16gScalingJoysDeltaArmRawValue : INT
GET
                    IF i16gScalingJoysDeltaArm.AppScalingMultiplier = 0 THEN
	_MatchLog^.Error("Get i16gScalingJoysDeltaArmRawValue", "Division by Zero!");
	RETURN;
End_IF

i16gScalingJoysDeltaArmRawValue := TO_INT((i16gScalingJoysDeltaArm.Value - i16gScalingJoysDeltaArm.AppScalingOffset) * i16gScalingJoysDeltaArm.AppScalingDivisor / i16gScalingJoysDeltaArm.AppScalingMultiplier);

                  
END_GET
END_PROPERTY

PROPERTY i16gScalingJoysArrowArmRawValue : INT
GET
                    IF i16gScalingJoysArrowArm.AppScalingMultiplier = 0 THEN
	_MatchLog^.Error("Get i16gScalingJoysArrowArmRawValue", "Division by Zero!");
	RETURN;
End_IF

i16gScalingJoysArrowArmRawValue := TO_INT((i16gScalingJoysArrowArm.Value - i16gScalingJoysArrowArm.AppScalingOffset) * i16gScalingJoysArrowArm.AppScalingDivisor / i16gScalingJoysArrowArm.AppScalingMultiplier);

                  
END_GET
END_PROPERTY

PROPERTY i16gScalingJoysTelescopeArmRawValue : INT
GET
                    IF i16gScalingJoysTelescopeArm.AppScalingMultiplier = 0 THEN
	_MatchLog^.Error("Get i16gScalingJoysTelescopeArmRawValue", "Division by Zero!");
	RETURN;
End_IF

i16gScalingJoysTelescopeArmRawValue := TO_INT((i16gScalingJoysTelescopeArm.Value - i16gScalingJoysTelescopeArm.AppScalingOffset) * i16gScalingJoysTelescopeArm.AppScalingDivisor / i16gScalingJoysTelescopeArm.AppScalingMultiplier);

                  
END_GET
END_PROPERTY

PROPERTY i16gScalingJoysTurretToolValue : INT
GET
                    IF i16gScalingJoysTurret.ToolScalingDivisor = 0 OR i16gScalingJoysTurret.AppScalingMultiplier = 0 THEN
	_MatchLog^.Error("Get i16gScalingJoysTurretToolValue", "Division by Zero!");
	RETURN;
END_IF

i16gScalingJoysTurretToolValue := TO_INT(((i16gScalingJoysTurret.Value - i16gScalingJoysTurret.AppScalingOffset) * i16gScalingJoysTurret.AppScalingDivisor / i16gScalingJoysTurret.AppScalingMultiplier * i16gScalingJoysTurret.ToolScalingMultiplier / i16gScalingJoysTurret.ToolScalingDivisor) + i16gScalingJoysTurret.ToolScalingOffset);

                  
END_GET
END_PROPERTY

PROPERTY i16gScalingJoysDeltaArmToolValue : INT
GET
                    IF i16gScalingJoysDeltaArm.ToolScalingDivisor = 0 OR i16gScalingJoysDeltaArm.AppScalingMultiplier = 0 THEN
	_MatchLog^.Error("Get i16gScalingJoysDeltaArmToolValue", "Division by Zero!");
	RETURN;
END_IF

i16gScalingJoysDeltaArmToolValue := TO_INT(((i16gScalingJoysDeltaArm.Value - i16gScalingJoysDeltaArm.AppScalingOffset) * i16gScalingJoysDeltaArm.AppScalingDivisor / i16gScalingJoysDeltaArm.AppScalingMultiplier * i16gScalingJoysDeltaArm.ToolScalingMultiplier / i16gScalingJoysDeltaArm.ToolScalingDivisor) + i16gScalingJoysDeltaArm.ToolScalingOffset);

                  
END_GET
END_PROPERTY

PROPERTY i16gScalingJoysArrowArmToolValue : INT
GET
                    IF i16gScalingJoysArrowArm.ToolScalingDivisor = 0 OR i16gScalingJoysArrowArm.AppScalingMultiplier = 0 THEN
	_MatchLog^.Error("Get i16gScalingJoysArrowArmToolValue", "Division by Zero!");
	RETURN;
END_IF

i16gScalingJoysArrowArmToolValue := TO_INT(((i16gScalingJoysArrowArm.Value - i16gScalingJoysArrowArm.AppScalingOffset) * i16gScalingJoysArrowArm.AppScalingDivisor / i16gScalingJoysArrowArm.AppScalingMultiplier * i16gScalingJoysArrowArm.ToolScalingMultiplier / i16gScalingJoysArrowArm.ToolScalingDivisor) + i16gScalingJoysArrowArm.ToolScalingOffset);

                  
END_GET
END_PROPERTY

PROPERTY i16gScalingJoysTelescopeArmToolValue : INT
GET
                    IF i16gScalingJoysTelescopeArm.ToolScalingDivisor = 0 OR i16gScalingJoysTelescopeArm.AppScalingMultiplier = 0 THEN
	_MatchLog^.Error("Get i16gScalingJoysTelescopeArmToolValue", "Division by Zero!");
	RETURN;
END_IF

i16gScalingJoysTelescopeArmToolValue := TO_INT(((i16gScalingJoysTelescopeArm.Value - i16gScalingJoysTelescopeArm.AppScalingOffset) * i16gScalingJoysTelescopeArm.AppScalingDivisor / i16gScalingJoysTelescopeArm.AppScalingMultiplier * i16gScalingJoysTelescopeArm.ToolScalingMultiplier / i16gScalingJoysTelescopeArm.ToolScalingDivisor) + i16gScalingJoysTelescopeArm.ToolScalingOffset);

                  
END_GET
END_PROPERTY

METHOD InitializeCanSignals
                  i16gScalingJoysTurret.AppScalingDivisor :=1;
i16gScalingJoysTurret.AppScalingMultiplier :=1;
i16gScalingJoysTurret.AppScalingOffset :=0;
i16gScalingJoysTurret.AppUnit :="";
i16gScalingJoysTurret.CanDefault :=0;
i16gScalingJoysTurret.CanInit :=0;
i16gScalingJoysTurret.CanMax :=VBasic.LibConst.I16_MAX;
i16gScalingJoysTurret.CanMin :=VBasic.LibConst.I16_MIN;
i16gScalingJoysTurret.CanUnit :="";
i16gScalingJoysTurret.Description :="new signal";
i16gScalingJoysTurret.ErrorReaction := eErrorReaction.ERSIG_DFLT;
i16gScalingJoysTurret.ReceiverAdress :=1;
i16gScalingJoysTurret.ToolScalingDivisor :=1;
i16gScalingJoysTurret.ToolScalingMultiplier :=1;
i16gScalingJoysTurret.ToolScalingOffset :=0;
i16gScalingJoysTurret.ToolUnit :="";

i16gScalingJoysDeltaArm.AppScalingDivisor :=1;
i16gScalingJoysDeltaArm.AppScalingMultiplier :=1;
i16gScalingJoysDeltaArm.AppScalingOffset :=0;
i16gScalingJoysDeltaArm.AppUnit :="";
i16gScalingJoysDeltaArm.CanDefault :=0;
i16gScalingJoysDeltaArm.CanInit :=0;
i16gScalingJoysDeltaArm.CanMax :=VBasic.LibConst.I16_MAX;
i16gScalingJoysDeltaArm.CanMin :=VBasic.LibConst.I16_MIN;
i16gScalingJoysDeltaArm.CanUnit :="";
i16gScalingJoysDeltaArm.Description :="new signal";
i16gScalingJoysDeltaArm.ErrorReaction := eErrorReaction.ERSIG_DFLT;
i16gScalingJoysDeltaArm.ReceiverAdress :=1;
i16gScalingJoysDeltaArm.ToolScalingDivisor :=1;
i16gScalingJoysDeltaArm.ToolScalingMultiplier :=1;
i16gScalingJoysDeltaArm.ToolScalingOffset :=0;
i16gScalingJoysDeltaArm.ToolUnit :="";

i16gScalingJoysArrowArm.AppScalingDivisor :=1;
i16gScalingJoysArrowArm.AppScalingMultiplier :=1;
i16gScalingJoysArrowArm.AppScalingOffset :=0;
i16gScalingJoysArrowArm.AppUnit :="";
i16gScalingJoysArrowArm.CanDefault :=0;
i16gScalingJoysArrowArm.CanInit :=0;
i16gScalingJoysArrowArm.CanMax :=VBasic.LibConst.I16_MAX;
i16gScalingJoysArrowArm.CanMin :=VBasic.LibConst.I16_MIN;
i16gScalingJoysArrowArm.CanUnit :="";
i16gScalingJoysArrowArm.Description :="new signal";
i16gScalingJoysArrowArm.ErrorReaction := eErrorReaction.ERSIG_DFLT;
i16gScalingJoysArrowArm.ReceiverAdress :=1;
i16gScalingJoysArrowArm.ToolScalingDivisor :=1;
i16gScalingJoysArrowArm.ToolScalingMultiplier :=1;
i16gScalingJoysArrowArm.ToolScalingOffset :=0;
i16gScalingJoysArrowArm.ToolUnit :="";

i16gScalingJoysTelescopeArm.AppScalingDivisor :=1;
i16gScalingJoysTelescopeArm.AppScalingMultiplier :=1;
i16gScalingJoysTelescopeArm.AppScalingOffset :=0;
i16gScalingJoysTelescopeArm.AppUnit :="";
i16gScalingJoysTelescopeArm.CanDefault :=0;
i16gScalingJoysTelescopeArm.CanInit :=0;
i16gScalingJoysTelescopeArm.CanMax :=VBasic.LibConst.I16_MAX;
i16gScalingJoysTelescopeArm.CanMin :=VBasic.LibConst.I16_MIN;
i16gScalingJoysTelescopeArm.CanUnit :="";
i16gScalingJoysTelescopeArm.Description :="new signal";
i16gScalingJoysTelescopeArm.ErrorReaction := eErrorReaction.ERSIG_DFLT;
i16gScalingJoysTelescopeArm.ReceiverAdress :=1;
i16gScalingJoysTelescopeArm.ToolScalingDivisor :=1;
i16gScalingJoysTelescopeArm.ToolScalingMultiplier :=1;
i16gScalingJoysTelescopeArm.ToolScalingOffset :=0;
i16gScalingJoysTelescopeArm.ToolUnit :="";


                
END_METHOD
END_FUNCTION_BLOCK

FUNCTION_BLOCK Msg12C1SendToEvision7MessageClass EXTENDS CanReceiveMessageClass
  VAR_INPUT
    u16gTelescopePVGValue : UInt16CanSignalClass;
    u16gTelescopeLengthPercentile : UInt16CanSignalClass;
    i16gGeneratorSolenoidValue : Int16CanSignalClass;
    i16gRPMSolenoidValue : Int16CanSignalClass;
    Counter : UInt32CanSignalClass;
  END_VAR

            
          

METHOD SetData
  VAR_INPUT
    CanMsgPointer : POINTER TO CanMessageClass;
  END_VAR
                  IF IsValidPointer(canMsgPointer,'SetData') THEN
	SUPER^.SetData(CanMsgPointer);
	//Set the new data
	u16gTelescopePVGValue.Value := canMsgPointer^.GetUint16(0);
	u16gTelescopeLengthPercentile.Value := canMsgPointer^.GetUint16(16);
	i16gGeneratorSolenoidValue.Value := canMsgPointer^.GetInt16(32);
	i16gRPMSolenoidValue.Value := canMsgPointer^.GetInt16(48);
	//And increase the counter
	Counter.Value := CanMsgPointer^.Counter.Value;
END_IF

                
END_METHOD

PROPERTY u16gTelescopePVGValueRawValue : UINT
GET
                    IF u16gTelescopePVGValue.AppScalingMultiplier = 0 THEN
	_MatchLog^.Error("Get u16gTelescopePVGValueRawValue", "Division by Zero!");
	RETURN;
End_IF

u16gTelescopePVGValueRawValue := TO_UINT((u16gTelescopePVGValue.Value - u16gTelescopePVGValue.AppScalingOffset) * u16gTelescopePVGValue.AppScalingDivisor / u16gTelescopePVGValue.AppScalingMultiplier);

                  
END_GET
END_PROPERTY

PROPERTY u16gTelescopeLengthPercentileRawValue : UINT
GET
                    IF u16gTelescopeLengthPercentile.AppScalingMultiplier = 0 THEN
	_MatchLog^.Error("Get u16gTelescopeLengthPercentileRawValue", "Division by Zero!");
	RETURN;
End_IF

u16gTelescopeLengthPercentileRawValue := TO_UINT((u16gTelescopeLengthPercentile.Value - u16gTelescopeLengthPercentile.AppScalingOffset) * u16gTelescopeLengthPercentile.AppScalingDivisor / u16gTelescopeLengthPercentile.AppScalingMultiplier);

                  
END_GET
END_PROPERTY

PROPERTY i16gGeneratorSolenoidValueRawValue : INT
GET
                    IF i16gGeneratorSolenoidValue.AppScalingMultiplier = 0 THEN
	_MatchLog^.Error("Get i16gGeneratorSolenoidValueRawValue", "Division by Zero!");
	RETURN;
End_IF

i16gGeneratorSolenoidValueRawValue := TO_INT((i16gGeneratorSolenoidValue.Value - i16gGeneratorSolenoidValue.AppScalingOffset) * i16gGeneratorSolenoidValue.AppScalingDivisor / i16gGeneratorSolenoidValue.AppScalingMultiplier);

                  
END_GET
END_PROPERTY

PROPERTY i16gRPMSolenoidValueRawValue : INT
GET
                    IF i16gRPMSolenoidValue.AppScalingMultiplier = 0 THEN
	_MatchLog^.Error("Get i16gRPMSolenoidValueRawValue", "Division by Zero!");
	RETURN;
End_IF

i16gRPMSolenoidValueRawValue := TO_INT((i16gRPMSolenoidValue.Value - i16gRPMSolenoidValue.AppScalingOffset) * i16gRPMSolenoidValue.AppScalingDivisor / i16gRPMSolenoidValue.AppScalingMultiplier);

                  
END_GET
END_PROPERTY

PROPERTY u16gTelescopePVGValueToolValue : UINT
GET
                    IF u16gTelescopePVGValue.ToolScalingDivisor = 0 OR u16gTelescopePVGValue.AppScalingMultiplier = 0 THEN
	_MatchLog^.Error("Get u16gTelescopePVGValueToolValue", "Division by Zero!");
	RETURN;
END_IF

u16gTelescopePVGValueToolValue := TO_UINT(((u16gTelescopePVGValue.Value - u16gTelescopePVGValue.AppScalingOffset) * u16gTelescopePVGValue.AppScalingDivisor / u16gTelescopePVGValue.AppScalingMultiplier * u16gTelescopePVGValue.ToolScalingMultiplier / u16gTelescopePVGValue.ToolScalingDivisor) + u16gTelescopePVGValue.ToolScalingOffset);

                  
END_GET
END_PROPERTY

PROPERTY u16gTelescopeLengthPercentileToolValue : UINT
GET
                    IF u16gTelescopeLengthPercentile.ToolScalingDivisor = 0 OR u16gTelescopeLengthPercentile.AppScalingMultiplier = 0 THEN
	_MatchLog^.Error("Get u16gTelescopeLengthPercentileToolValue", "Division by Zero!");
	RETURN;
END_IF

u16gTelescopeLengthPercentileToolValue := TO_UINT(((u16gTelescopeLengthPercentile.Value - u16gTelescopeLengthPercentile.AppScalingOffset) * u16gTelescopeLengthPercentile.AppScalingDivisor / u16gTelescopeLengthPercentile.AppScalingMultiplier * u16gTelescopeLengthPercentile.ToolScalingMultiplier / u16gTelescopeLengthPercentile.ToolScalingDivisor) + u16gTelescopeLengthPercentile.ToolScalingOffset);

                  
END_GET
END_PROPERTY

PROPERTY i16gGeneratorSolenoidValueToolValue : INT
GET
                    IF i16gGeneratorSolenoidValue.ToolScalingDivisor = 0 OR i16gGeneratorSolenoidValue.AppScalingMultiplier = 0 THEN
	_MatchLog^.Error("Get i16gGeneratorSolenoidValueToolValue", "Division by Zero!");
	RETURN;
END_IF

i16gGeneratorSolenoidValueToolValue := TO_INT(((i16gGeneratorSolenoidValue.Value - i16gGeneratorSolenoidValue.AppScalingOffset) * i16gGeneratorSolenoidValue.AppScalingDivisor / i16gGeneratorSolenoidValue.AppScalingMultiplier * i16gGeneratorSolenoidValue.ToolScalingMultiplier / i16gGeneratorSolenoidValue.ToolScalingDivisor) + i16gGeneratorSolenoidValue.ToolScalingOffset);

                  
END_GET
END_PROPERTY

PROPERTY i16gRPMSolenoidValueToolValue : INT
GET
                    IF i16gRPMSolenoidValue.ToolScalingDivisor = 0 OR i16gRPMSolenoidValue.AppScalingMultiplier = 0 THEN
	_MatchLog^.Error("Get i16gRPMSolenoidValueToolValue", "Division by Zero!");
	RETURN;
END_IF

i16gRPMSolenoidValueToolValue := TO_INT(((i16gRPMSolenoidValue.Value - i16gRPMSolenoidValue.AppScalingOffset) * i16gRPMSolenoidValue.AppScalingDivisor / i16gRPMSolenoidValue.AppScalingMultiplier * i16gRPMSolenoidValue.ToolScalingMultiplier / i16gRPMSolenoidValue.ToolScalingDivisor) + i16gRPMSolenoidValue.ToolScalingOffset);

                  
END_GET
END_PROPERTY

METHOD InitializeCanSignals
                  u16gTelescopePVGValue.AppScalingDivisor :=1;
u16gTelescopePVGValue.AppScalingMultiplier :=1;
u16gTelescopePVGValue.AppScalingOffset :=0;
u16gTelescopePVGValue.AppUnit :="";
u16gTelescopePVGValue.CanDefault :=0;
u16gTelescopePVGValue.CanInit :=0;
u16gTelescopePVGValue.CanMax :=VBasic.LibConst.U16_MAX;
u16gTelescopePVGValue.CanMin :=VBasic.LibConst.U16_MIN;
u16gTelescopePVGValue.CanUnit :="";
u16gTelescopePVGValue.Description :="new signal";
u16gTelescopePVGValue.ErrorReaction := eErrorReaction.ERSIG_DFLT;
u16gTelescopePVGValue.ReceiverAdress :=1;
u16gTelescopePVGValue.ToolScalingDivisor :=1;
u16gTelescopePVGValue.ToolScalingMultiplier :=1;
u16gTelescopePVGValue.ToolScalingOffset :=0;
u16gTelescopePVGValue.ToolUnit :="";

u16gTelescopeLengthPercentile.AppScalingDivisor :=1;
u16gTelescopeLengthPercentile.AppScalingMultiplier :=1;
u16gTelescopeLengthPercentile.AppScalingOffset :=0;
u16gTelescopeLengthPercentile.AppUnit :="";
u16gTelescopeLengthPercentile.CanDefault :=0;
u16gTelescopeLengthPercentile.CanInit :=0;
u16gTelescopeLengthPercentile.CanMax :=VBasic.LibConst.U16_MAX;
u16gTelescopeLengthPercentile.CanMin :=VBasic.LibConst.U16_MIN;
u16gTelescopeLengthPercentile.CanUnit :="";
u16gTelescopeLengthPercentile.Description :="new signal";
u16gTelescopeLengthPercentile.ErrorReaction := eErrorReaction.ERSIG_DFLT;
u16gTelescopeLengthPercentile.ReceiverAdress :=1;
u16gTelescopeLengthPercentile.ToolScalingDivisor :=1;
u16gTelescopeLengthPercentile.ToolScalingMultiplier :=1;
u16gTelescopeLengthPercentile.ToolScalingOffset :=0;
u16gTelescopeLengthPercentile.ToolUnit :="";

i16gGeneratorSolenoidValue.AppScalingDivisor :=1;
i16gGeneratorSolenoidValue.AppScalingMultiplier :=1;
i16gGeneratorSolenoidValue.AppScalingOffset :=0;
i16gGeneratorSolenoidValue.AppUnit :="";
i16gGeneratorSolenoidValue.CanDefault :=0;
i16gGeneratorSolenoidValue.CanInit :=0;
i16gGeneratorSolenoidValue.CanMax :=VBasic.LibConst.I16_MAX;
i16gGeneratorSolenoidValue.CanMin :=VBasic.LibConst.I16_MIN;
i16gGeneratorSolenoidValue.CanUnit :="";
i16gGeneratorSolenoidValue.Description :="new signal";
i16gGeneratorSolenoidValue.ErrorReaction := eErrorReaction.ERSIG_DFLT;
i16gGeneratorSolenoidValue.ReceiverAdress :=1;
i16gGeneratorSolenoidValue.ToolScalingDivisor :=1;
i16gGeneratorSolenoidValue.ToolScalingMultiplier :=1;
i16gGeneratorSolenoidValue.ToolScalingOffset :=0;
i16gGeneratorSolenoidValue.ToolUnit :="";

i16gRPMSolenoidValue.AppScalingDivisor :=1;
i16gRPMSolenoidValue.AppScalingMultiplier :=1;
i16gRPMSolenoidValue.AppScalingOffset :=0;
i16gRPMSolenoidValue.AppUnit :="";
i16gRPMSolenoidValue.CanDefault :=0;
i16gRPMSolenoidValue.CanInit :=0;
i16gRPMSolenoidValue.CanMax :=VBasic.LibConst.I16_MAX;
i16gRPMSolenoidValue.CanMin :=VBasic.LibConst.I16_MIN;
i16gRPMSolenoidValue.CanUnit :="";
i16gRPMSolenoidValue.Description :="new signal";
i16gRPMSolenoidValue.ErrorReaction := eErrorReaction.ERSIG_DFLT;
i16gRPMSolenoidValue.ReceiverAdress :=1;
i16gRPMSolenoidValue.ToolScalingDivisor :=1;
i16gRPMSolenoidValue.ToolScalingMultiplier :=1;
i16gRPMSolenoidValue.ToolScalingOffset :=0;
i16gRPMSolenoidValue.ToolUnit :="";


                
END_METHOD
END_FUNCTION_BLOCK

FUNCTION_BLOCK Msg13C1SendToEvision7MessageClass EXTENDS CanReceiveMessageClass
  VAR_INPUT
    i16gBypassPressureSensorValue : Int16CanSignalClass;
    u16gBatteryVoltageMv : UInt16CanSignalClass;
    u16RemainingRegenTimeAverage : UInt16CanSignalClass;
    boElectricMotorForbidden : BoolCanSignalClass;
    boReloadWithGeneratorOn : BoolCanSignalClass;
    boPictoColdOilTankTemperature : BoolCanSignalClass;
    boPictoWarningValidCycleMast : BoolCanSignalClass;
    Counter : UInt32CanSignalClass;
  END_VAR

            
          

METHOD SetData
  VAR_INPUT
    CanMsgPointer : POINTER TO CanMessageClass;
  END_VAR
                  IF IsValidPointer(canMsgPointer,'SetData') THEN
	SUPER^.SetData(CanMsgPointer);
	//Set the new data
	i16gBypassPressureSensorValue.Value := canMsgPointer^.GetInt16(0);
	u16gBatteryVoltageMv.Value := canMsgPointer^.GetUint16(16);
	u16RemainingRegenTimeAverage.Value := canMsgPointer^.GetUint16(32);
	boElectricMotorForbidden.Value := canMsgPointer^.GetBoolOnBit(48);
	boReloadWithGeneratorOn.Value := canMsgPointer^.GetBoolOnBit(49);
	boPictoColdOilTankTemperature.Value := canMsgPointer^.GetBoolOnBit(50);
	boPictoWarningValidCycleMast.Value := canMsgPointer^.GetBoolOnBit(51);
	//And increase the counter
	Counter.Value := CanMsgPointer^.Counter.Value;
END_IF

                
END_METHOD

PROPERTY i16gBypassPressureSensorValueRawValue : INT
GET
                    IF i16gBypassPressureSensorValue.AppScalingMultiplier = 0 THEN
	_MatchLog^.Error("Get i16gBypassPressureSensorValueRawValue", "Division by Zero!");
	RETURN;
End_IF

i16gBypassPressureSensorValueRawValue := TO_INT((i16gBypassPressureSensorValue.Value - i16gBypassPressureSensorValue.AppScalingOffset) * i16gBypassPressureSensorValue.AppScalingDivisor / i16gBypassPressureSensorValue.AppScalingMultiplier);

                  
END_GET
END_PROPERTY

PROPERTY u16gBatteryVoltageMvRawValue : UINT
GET
                    IF u16gBatteryVoltageMv.AppScalingMultiplier = 0 THEN
	_MatchLog^.Error("Get u16gBatteryVoltageMvRawValue", "Division by Zero!");
	RETURN;
End_IF

u16gBatteryVoltageMvRawValue := TO_UINT((u16gBatteryVoltageMv.Value - u16gBatteryVoltageMv.AppScalingOffset) * u16gBatteryVoltageMv.AppScalingDivisor / u16gBatteryVoltageMv.AppScalingMultiplier);

                  
END_GET
END_PROPERTY

PROPERTY u16RemainingRegenTimeAverageRawValue : UINT
GET
                    IF u16RemainingRegenTimeAverage.AppScalingMultiplier = 0 THEN
	_MatchLog^.Error("Get u16RemainingRegenTimeAverageRawValue", "Division by Zero!");
	RETURN;
End_IF

u16RemainingRegenTimeAverageRawValue := TO_UINT((u16RemainingRegenTimeAverage.Value - u16RemainingRegenTimeAverage.AppScalingOffset) * u16RemainingRegenTimeAverage.AppScalingDivisor / u16RemainingRegenTimeAverage.AppScalingMultiplier);

                  
END_GET
END_PROPERTY

PROPERTY boElectricMotorForbiddenRawValue : BOOL
GET
                    boElectricMotorForbiddenRawValue := boElectricMotorForbidden.Value;

                  
END_GET
END_PROPERTY

PROPERTY boReloadWithGeneratorOnRawValue : BOOL
GET
                    boReloadWithGeneratorOnRawValue := boReloadWithGeneratorOn.Value;

                  
END_GET
END_PROPERTY

PROPERTY boPictoColdOilTankTemperatureRawValue : BOOL
GET
                    boPictoColdOilTankTemperatureRawValue := boPictoColdOilTankTemperature.Value;

                  
END_GET
END_PROPERTY

PROPERTY boPictoWarningValidCycleMastRawValue : BOOL
GET
                    boPictoWarningValidCycleMastRawValue := boPictoWarningValidCycleMast.Value;

                  
END_GET
END_PROPERTY

PROPERTY i16gBypassPressureSensorValueToolValue : INT
GET
                    IF i16gBypassPressureSensorValue.ToolScalingDivisor = 0 OR i16gBypassPressureSensorValue.AppScalingMultiplier = 0 THEN
	_MatchLog^.Error("Get i16gBypassPressureSensorValueToolValue", "Division by Zero!");
	RETURN;
END_IF

i16gBypassPressureSensorValueToolValue := TO_INT(((i16gBypassPressureSensorValue.Value - i16gBypassPressureSensorValue.AppScalingOffset) * i16gBypassPressureSensorValue.AppScalingDivisor / i16gBypassPressureSensorValue.AppScalingMultiplier * i16gBypassPressureSensorValue.ToolScalingMultiplier / i16gBypassPressureSensorValue.ToolScalingDivisor) + i16gBypassPressureSensorValue.ToolScalingOffset);

                  
END_GET
END_PROPERTY

PROPERTY u16gBatteryVoltageMvToolValue : UINT
GET
                    IF u16gBatteryVoltageMv.ToolScalingDivisor = 0 OR u16gBatteryVoltageMv.AppScalingMultiplier = 0 THEN
	_MatchLog^.Error("Get u16gBatteryVoltageMvToolValue", "Division by Zero!");
	RETURN;
END_IF

u16gBatteryVoltageMvToolValue := TO_UINT(((u16gBatteryVoltageMv.Value - u16gBatteryVoltageMv.AppScalingOffset) * u16gBatteryVoltageMv.AppScalingDivisor / u16gBatteryVoltageMv.AppScalingMultiplier * u16gBatteryVoltageMv.ToolScalingMultiplier / u16gBatteryVoltageMv.ToolScalingDivisor) + u16gBatteryVoltageMv.ToolScalingOffset);

                  
END_GET
END_PROPERTY

PROPERTY u16RemainingRegenTimeAverageToolValue : UINT
GET
                    IF u16RemainingRegenTimeAverage.ToolScalingDivisor = 0 OR u16RemainingRegenTimeAverage.AppScalingMultiplier = 0 THEN
	_MatchLog^.Error("Get u16RemainingRegenTimeAverageToolValue", "Division by Zero!");
	RETURN;
END_IF

u16RemainingRegenTimeAverageToolValue := TO_UINT(((u16RemainingRegenTimeAverage.Value - u16RemainingRegenTimeAverage.AppScalingOffset) * u16RemainingRegenTimeAverage.AppScalingDivisor / u16RemainingRegenTimeAverage.AppScalingMultiplier * u16RemainingRegenTimeAverage.ToolScalingMultiplier / u16RemainingRegenTimeAverage.ToolScalingDivisor) + u16RemainingRegenTimeAverage.ToolScalingOffset);

                  
END_GET
END_PROPERTY

PROPERTY boElectricMotorForbiddenToolValue : BOOL
GET
                    boElectricMotorForbiddenToolValue := boElectricMotorForbidden.Value;

                  
END_GET
END_PROPERTY

PROPERTY boReloadWithGeneratorOnToolValue : BOOL
GET
                    boReloadWithGeneratorOnToolValue := boReloadWithGeneratorOn.Value;

                  
END_GET
END_PROPERTY

PROPERTY boPictoColdOilTankTemperatureToolValue : BOOL
GET
                    boPictoColdOilTankTemperatureToolValue := boPictoColdOilTankTemperature.Value;

                  
END_GET
END_PROPERTY

PROPERTY boPictoWarningValidCycleMastToolValue : BOOL
GET
                    boPictoWarningValidCycleMastToolValue := boPictoWarningValidCycleMast.Value;

                  
END_GET
END_PROPERTY

METHOD InitializeCanSignals
                  i16gBypassPressureSensorValue.AppScalingDivisor :=1;
i16gBypassPressureSensorValue.AppScalingMultiplier :=1;
i16gBypassPressureSensorValue.AppScalingOffset :=0;
i16gBypassPressureSensorValue.AppUnit :="";
i16gBypassPressureSensorValue.CanDefault :=0;
i16gBypassPressureSensorValue.CanInit :=0;
i16gBypassPressureSensorValue.CanMax :=VBasic.LibConst.I16_MAX;
i16gBypassPressureSensorValue.CanMin :=VBasic.LibConst.I16_MIN;
i16gBypassPressureSensorValue.CanUnit :="";
i16gBypassPressureSensorValue.Description :="new signal";
i16gBypassPressureSensorValue.ErrorReaction := eErrorReaction.ERSIG_DFLT;
i16gBypassPressureSensorValue.ReceiverAdress :=1;
i16gBypassPressureSensorValue.ToolScalingDivisor :=1;
i16gBypassPressureSensorValue.ToolScalingMultiplier :=1;
i16gBypassPressureSensorValue.ToolScalingOffset :=0;
i16gBypassPressureSensorValue.ToolUnit :="";

u16gBatteryVoltageMv.AppScalingDivisor :=1;
u16gBatteryVoltageMv.AppScalingMultiplier :=1;
u16gBatteryVoltageMv.AppScalingOffset :=0;
u16gBatteryVoltageMv.AppUnit :="";
u16gBatteryVoltageMv.CanDefault :=0;
u16gBatteryVoltageMv.CanInit :=0;
u16gBatteryVoltageMv.CanMax :=VBasic.LibConst.U16_MAX;
u16gBatteryVoltageMv.CanMin :=VBasic.LibConst.U16_MIN;
u16gBatteryVoltageMv.CanUnit :="";
u16gBatteryVoltageMv.Description :="new signal";
u16gBatteryVoltageMv.ErrorReaction := eErrorReaction.ERSIG_DFLT;
u16gBatteryVoltageMv.ReceiverAdress :=1;
u16gBatteryVoltageMv.ToolScalingDivisor :=1;
u16gBatteryVoltageMv.ToolScalingMultiplier :=1;
u16gBatteryVoltageMv.ToolScalingOffset :=0;
u16gBatteryVoltageMv.ToolUnit :="";

u16RemainingRegenTimeAverage.AppScalingDivisor :=1;
u16RemainingRegenTimeAverage.AppScalingMultiplier :=1;
u16RemainingRegenTimeAverage.AppScalingOffset :=0;
u16RemainingRegenTimeAverage.AppUnit :="";
u16RemainingRegenTimeAverage.CanDefault :=0;
u16RemainingRegenTimeAverage.CanInit :=0;
u16RemainingRegenTimeAverage.CanMax :=VBasic.LibConst.U16_MAX;
u16RemainingRegenTimeAverage.CanMin :=VBasic.LibConst.U16_MIN;
u16RemainingRegenTimeAverage.CanUnit :="";
u16RemainingRegenTimeAverage.Description :="new signal";
u16RemainingRegenTimeAverage.ErrorReaction := eErrorReaction.ERSIG_DFLT;
u16RemainingRegenTimeAverage.ReceiverAdress :=1;
u16RemainingRegenTimeAverage.ToolScalingDivisor :=1;
u16RemainingRegenTimeAverage.ToolScalingMultiplier :=1;
u16RemainingRegenTimeAverage.ToolScalingOffset :=0;
u16RemainingRegenTimeAverage.ToolUnit :="";

boElectricMotorForbidden.AppScalingDivisor :=1;
boElectricMotorForbidden.AppScalingMultiplier :=1;
boElectricMotorForbidden.AppScalingOffset :=0;
boElectricMotorForbidden.AppUnit :="";
boElectricMotorForbidden.CanDefault :=0;
boElectricMotorForbidden.CanInit :=0;
boElectricMotorForbidden.CanMax :=1;
boElectricMotorForbidden.CanMin :=0;
boElectricMotorForbidden.CanUnit :="";
boElectricMotorForbidden.Description :="new signal";
boElectricMotorForbidden.ErrorReaction := eErrorReaction.ERSIG_DFLT;
boElectricMotorForbidden.ReceiverAdress :=1;
boElectricMotorForbidden.ToolScalingDivisor :=1;
boElectricMotorForbidden.ToolScalingMultiplier :=1;
boElectricMotorForbidden.ToolScalingOffset :=0;
boElectricMotorForbidden.ToolUnit :="";

boReloadWithGeneratorOn.AppScalingDivisor :=1;
boReloadWithGeneratorOn.AppScalingMultiplier :=1;
boReloadWithGeneratorOn.AppScalingOffset :=0;
boReloadWithGeneratorOn.AppUnit :="";
boReloadWithGeneratorOn.CanDefault :=0;
boReloadWithGeneratorOn.CanInit :=0;
boReloadWithGeneratorOn.CanMax :=1;
boReloadWithGeneratorOn.CanMin :=0;
boReloadWithGeneratorOn.CanUnit :="";
boReloadWithGeneratorOn.Description :="new signal";
boReloadWithGeneratorOn.ErrorReaction := eErrorReaction.ERSIG_DFLT;
boReloadWithGeneratorOn.ReceiverAdress :=1;
boReloadWithGeneratorOn.ToolScalingDivisor :=1;
boReloadWithGeneratorOn.ToolScalingMultiplier :=1;
boReloadWithGeneratorOn.ToolScalingOffset :=0;
boReloadWithGeneratorOn.ToolUnit :="";

boPictoColdOilTankTemperature.AppScalingDivisor :=1;
boPictoColdOilTankTemperature.AppScalingMultiplier :=1;
boPictoColdOilTankTemperature.AppScalingOffset :=0;
boPictoColdOilTankTemperature.AppUnit :="";
boPictoColdOilTankTemperature.CanDefault :=0;
boPictoColdOilTankTemperature.CanInit :=0;
boPictoColdOilTankTemperature.CanMax :=1;
boPictoColdOilTankTemperature.CanMin :=0;
boPictoColdOilTankTemperature.CanUnit :="";
boPictoColdOilTankTemperature.Description :="new signal";
boPictoColdOilTankTemperature.ErrorReaction := eErrorReaction.ERSIG_DFLT;
boPictoColdOilTankTemperature.ReceiverAdress :=1;
boPictoColdOilTankTemperature.ToolScalingDivisor :=1;
boPictoColdOilTankTemperature.ToolScalingMultiplier :=1;
boPictoColdOilTankTemperature.ToolScalingOffset :=0;
boPictoColdOilTankTemperature.ToolUnit :="";

boPictoWarningValidCycleMast.AppScalingDivisor :=1;
boPictoWarningValidCycleMast.AppScalingMultiplier :=1;
boPictoWarningValidCycleMast.AppScalingOffset :=0;
boPictoWarningValidCycleMast.AppUnit :="";
boPictoWarningValidCycleMast.CanDefault :=0;
boPictoWarningValidCycleMast.CanInit :=0;
boPictoWarningValidCycleMast.CanMax :=1;
boPictoWarningValidCycleMast.CanMin :=0;
boPictoWarningValidCycleMast.CanUnit :="";
boPictoWarningValidCycleMast.Description :="new signal";
boPictoWarningValidCycleMast.ErrorReaction := eErrorReaction.ERSIG_DFLT;
boPictoWarningValidCycleMast.ReceiverAdress :=1;
boPictoWarningValidCycleMast.ToolScalingDivisor :=1;
boPictoWarningValidCycleMast.ToolScalingMultiplier :=1;
boPictoWarningValidCycleMast.ToolScalingOffset :=0;
boPictoWarningValidCycleMast.ToolUnit :="";


                
END_METHOD
END_FUNCTION_BLOCK

FUNCTION_BLOCK Msg14C1SendToEvision7MessageClass EXTENDS CanReceiveMessageClass
  VAR_INPUT
    i16OilTankTemperatureValue : Int16CanSignalClass;
    u16TotalRegenHours : UInt16CanSignalClass;
    u16TotalElectricHours : UInt16CanSignalClass;
    Counter : UInt32CanSignalClass;
  END_VAR

            
          

METHOD SetData
  VAR_INPUT
    CanMsgPointer : POINTER TO CanMessageClass;
  END_VAR
                  IF IsValidPointer(canMsgPointer,'SetData') THEN
	SUPER^.SetData(CanMsgPointer);
	//Set the new data
	i16OilTankTemperatureValue.Value := canMsgPointer^.GetInt16(0);
	u16TotalRegenHours.Value := canMsgPointer^.GetUint16(16);
	u16TotalElectricHours.Value := canMsgPointer^.GetUint16(32);
	//And increase the counter
	Counter.Value := CanMsgPointer^.Counter.Value;
END_IF

                
END_METHOD

PROPERTY i16OilTankTemperatureValueRawValue : INT
GET
                    IF i16OilTankTemperatureValue.AppScalingMultiplier = 0 THEN
	_MatchLog^.Error("Get i16OilTankTemperatureValueRawValue", "Division by Zero!");
	RETURN;
End_IF

i16OilTankTemperatureValueRawValue := TO_INT((i16OilTankTemperatureValue.Value - i16OilTankTemperatureValue.AppScalingOffset) * i16OilTankTemperatureValue.AppScalingDivisor / i16OilTankTemperatureValue.AppScalingMultiplier);

                  
END_GET
END_PROPERTY

PROPERTY u16TotalRegenHoursRawValue : UINT
GET
                    IF u16TotalRegenHours.AppScalingMultiplier = 0 THEN
	_MatchLog^.Error("Get u16TotalRegenHoursRawValue", "Division by Zero!");
	RETURN;
End_IF

u16TotalRegenHoursRawValue := TO_UINT((u16TotalRegenHours.Value - u16TotalRegenHours.AppScalingOffset) * u16TotalRegenHours.AppScalingDivisor / u16TotalRegenHours.AppScalingMultiplier);

                  
END_GET
END_PROPERTY

PROPERTY u16TotalElectricHoursRawValue : UINT
GET
                    IF u16TotalElectricHours.AppScalingMultiplier = 0 THEN
	_MatchLog^.Error("Get u16TotalElectricHoursRawValue", "Division by Zero!");
	RETURN;
End_IF

u16TotalElectricHoursRawValue := TO_UINT((u16TotalElectricHours.Value - u16TotalElectricHours.AppScalingOffset) * u16TotalElectricHours.AppScalingDivisor / u16TotalElectricHours.AppScalingMultiplier);

                  
END_GET
END_PROPERTY

PROPERTY i16OilTankTemperatureValueToolValue : INT
GET
                    IF i16OilTankTemperatureValue.ToolScalingDivisor = 0 OR i16OilTankTemperatureValue.AppScalingMultiplier = 0 THEN
	_MatchLog^.Error("Get i16OilTankTemperatureValueToolValue", "Division by Zero!");
	RETURN;
END_IF

i16OilTankTemperatureValueToolValue := TO_INT(((i16OilTankTemperatureValue.Value - i16OilTankTemperatureValue.AppScalingOffset) * i16OilTankTemperatureValue.AppScalingDivisor / i16OilTankTemperatureValue.AppScalingMultiplier * i16OilTankTemperatureValue.ToolScalingMultiplier / i16OilTankTemperatureValue.ToolScalingDivisor) + i16OilTankTemperatureValue.ToolScalingOffset);

                  
END_GET
END_PROPERTY

PROPERTY u16TotalRegenHoursToolValue : UINT
GET
                    IF u16TotalRegenHours.ToolScalingDivisor = 0 OR u16TotalRegenHours.AppScalingMultiplier = 0 THEN
	_MatchLog^.Error("Get u16TotalRegenHoursToolValue", "Division by Zero!");
	RETURN;
END_IF

u16TotalRegenHoursToolValue := TO_UINT(((u16TotalRegenHours.Value - u16TotalRegenHours.AppScalingOffset) * u16TotalRegenHours.AppScalingDivisor / u16TotalRegenHours.AppScalingMultiplier * u16TotalRegenHours.ToolScalingMultiplier / u16TotalRegenHours.ToolScalingDivisor) + u16TotalRegenHours.ToolScalingOffset);

                  
END_GET
END_PROPERTY

PROPERTY u16TotalElectricHoursToolValue : UINT
GET
                    IF u16TotalElectricHours.ToolScalingDivisor = 0 OR u16TotalElectricHours.AppScalingMultiplier = 0 THEN
	_MatchLog^.Error("Get u16TotalElectricHoursToolValue", "Division by Zero!");
	RETURN;
END_IF

u16TotalElectricHoursToolValue := TO_UINT(((u16TotalElectricHours.Value - u16TotalElectricHours.AppScalingOffset) * u16TotalElectricHours.AppScalingDivisor / u16TotalElectricHours.AppScalingMultiplier * u16TotalElectricHours.ToolScalingMultiplier / u16TotalElectricHours.ToolScalingDivisor) + u16TotalElectricHours.ToolScalingOffset);

                  
END_GET
END_PROPERTY

METHOD InitializeCanSignals
                  i16OilTankTemperatureValue.AppScalingDivisor :=1;
i16OilTankTemperatureValue.AppScalingMultiplier :=1;
i16OilTankTemperatureValue.AppScalingOffset :=0;
i16OilTankTemperatureValue.AppUnit :="";
i16OilTankTemperatureValue.CanDefault :=0;
i16OilTankTemperatureValue.CanInit :=0;
i16OilTankTemperatureValue.CanMax :=VBasic.LibConst.I16_MAX;
i16OilTankTemperatureValue.CanMin :=VBasic.LibConst.I16_MIN;
i16OilTankTemperatureValue.CanUnit :="";
i16OilTankTemperatureValue.Description :="new signal";
i16OilTankTemperatureValue.ErrorReaction := eErrorReaction.ERSIG_DFLT;
i16OilTankTemperatureValue.ReceiverAdress :=1;
i16OilTankTemperatureValue.ToolScalingDivisor :=1;
i16OilTankTemperatureValue.ToolScalingMultiplier :=1;
i16OilTankTemperatureValue.ToolScalingOffset :=0;
i16OilTankTemperatureValue.ToolUnit :="";

u16TotalRegenHours.AppScalingDivisor :=1;
u16TotalRegenHours.AppScalingMultiplier :=1;
u16TotalRegenHours.AppScalingOffset :=0;
u16TotalRegenHours.AppUnit :="";
u16TotalRegenHours.CanDefault :=0;
u16TotalRegenHours.CanInit :=0;
u16TotalRegenHours.CanMax :=VBasic.LibConst.U16_MAX;
u16TotalRegenHours.CanMin :=VBasic.LibConst.U16_MIN;
u16TotalRegenHours.CanUnit :="";
u16TotalRegenHours.Description :="new signal";
u16TotalRegenHours.ErrorReaction := eErrorReaction.ERSIG_DFLT;
u16TotalRegenHours.ReceiverAdress :=1;
u16TotalRegenHours.ToolScalingDivisor :=1;
u16TotalRegenHours.ToolScalingMultiplier :=1;
u16TotalRegenHours.ToolScalingOffset :=0;
u16TotalRegenHours.ToolUnit :="";

u16TotalElectricHours.AppScalingDivisor :=1;
u16TotalElectricHours.AppScalingMultiplier :=1;
u16TotalElectricHours.AppScalingOffset :=0;
u16TotalElectricHours.AppUnit :="";
u16TotalElectricHours.CanDefault :=0;
u16TotalElectricHours.CanInit :=0;
u16TotalElectricHours.CanMax :=VBasic.LibConst.U16_MAX;
u16TotalElectricHours.CanMin :=VBasic.LibConst.U16_MIN;
u16TotalElectricHours.CanUnit :="";
u16TotalElectricHours.Description :="new signal";
u16TotalElectricHours.ErrorReaction := eErrorReaction.ERSIG_DFLT;
u16TotalElectricHours.ReceiverAdress :=1;
u16TotalElectricHours.ToolScalingDivisor :=1;
u16TotalElectricHours.ToolScalingMultiplier :=1;
u16TotalElectricHours.ToolScalingOffset :=0;
u16TotalElectricHours.ToolUnit :="";


                
END_METHOD
END_FUNCTION_BLOCK

FUNCTION_BLOCK MsgDebugC1SendToEvision7MessageClass EXTENDS CanReceiveMessageClass
  VAR_INPUT
    u16FaultyValue : UInt16CanSignalClass;
    u8DeviceNum : UInt8CanSignalClass;
    u8ErrorCode : UInt8CanSignalClass;
    i16DebugVehicleSlope : Int16CanSignalClass;
    Counter : UInt32CanSignalClass;
  END_VAR

            
          

METHOD SetData
  VAR_INPUT
    CanMsgPointer : POINTER TO CanMessageClass;
  END_VAR
                  IF IsValidPointer(canMsgPointer,'SetData') THEN
	SUPER^.SetData(CanMsgPointer);
	//Set the new data
	u16FaultyValue.Value := canMsgPointer^.GetUint16(0);
	u8DeviceNum.Value := canMsgPointer^.GetUint8(16);
	u8ErrorCode.Value := canMsgPointer^.GetUint8(24);
	i16DebugVehicleSlope.Value := canMsgPointer^.GetInt16(32);
	//And increase the counter
	Counter.Value := CanMsgPointer^.Counter.Value;
END_IF

                
END_METHOD

PROPERTY u16FaultyValueRawValue : UINT
GET
                    IF u16FaultyValue.AppScalingMultiplier = 0 THEN
	_MatchLog^.Error("Get u16FaultyValueRawValue", "Division by Zero!");
	RETURN;
End_IF

u16FaultyValueRawValue := TO_UINT((u16FaultyValue.Value - u16FaultyValue.AppScalingOffset) * u16FaultyValue.AppScalingDivisor / u16FaultyValue.AppScalingMultiplier);

                  
END_GET
END_PROPERTY

PROPERTY u8DeviceNumRawValue : USINT
GET
                    IF u8DeviceNum.AppScalingMultiplier = 0 THEN
	_MatchLog^.Error("Get u8DeviceNumRawValue", "Division by Zero!");
	RETURN;
End_IF

u8DeviceNumRawValue := TO_USINT((u8DeviceNum.Value - u8DeviceNum.AppScalingOffset) * u8DeviceNum.AppScalingDivisor / u8DeviceNum.AppScalingMultiplier);

                  
END_GET
END_PROPERTY

PROPERTY u8ErrorCodeRawValue : USINT
GET
                    IF u8ErrorCode.AppScalingMultiplier = 0 THEN
	_MatchLog^.Error("Get u8ErrorCodeRawValue", "Division by Zero!");
	RETURN;
End_IF

u8ErrorCodeRawValue := TO_USINT((u8ErrorCode.Value - u8ErrorCode.AppScalingOffset) * u8ErrorCode.AppScalingDivisor / u8ErrorCode.AppScalingMultiplier);

                  
END_GET
END_PROPERTY

PROPERTY i16DebugVehicleSlopeRawValue : INT
GET
                    IF i16DebugVehicleSlope.AppScalingMultiplier = 0 THEN
	_MatchLog^.Error("Get i16DebugVehicleSlopeRawValue", "Division by Zero!");
	RETURN;
End_IF

i16DebugVehicleSlopeRawValue := TO_INT((i16DebugVehicleSlope.Value - i16DebugVehicleSlope.AppScalingOffset) * i16DebugVehicleSlope.AppScalingDivisor / i16DebugVehicleSlope.AppScalingMultiplier);

                  
END_GET
END_PROPERTY

PROPERTY u16FaultyValueToolValue : UINT
GET
                    IF u16FaultyValue.ToolScalingDivisor = 0 OR u16FaultyValue.AppScalingMultiplier = 0 THEN
	_MatchLog^.Error("Get u16FaultyValueToolValue", "Division by Zero!");
	RETURN;
END_IF

u16FaultyValueToolValue := TO_UINT(((u16FaultyValue.Value - u16FaultyValue.AppScalingOffset) * u16FaultyValue.AppScalingDivisor / u16FaultyValue.AppScalingMultiplier * u16FaultyValue.ToolScalingMultiplier / u16FaultyValue.ToolScalingDivisor) + u16FaultyValue.ToolScalingOffset);

                  
END_GET
END_PROPERTY

PROPERTY u8DeviceNumToolValue : USINT
GET
                    IF u8DeviceNum.ToolScalingDivisor = 0 OR u8DeviceNum.AppScalingMultiplier = 0 THEN
	_MatchLog^.Error("Get u8DeviceNumToolValue", "Division by Zero!");
	RETURN;
END_IF

u8DeviceNumToolValue := TO_USINT(((u8DeviceNum.Value - u8DeviceNum.AppScalingOffset) * u8DeviceNum.AppScalingDivisor / u8DeviceNum.AppScalingMultiplier * u8DeviceNum.ToolScalingMultiplier / u8DeviceNum.ToolScalingDivisor) + u8DeviceNum.ToolScalingOffset);

                  
END_GET
END_PROPERTY

PROPERTY u8ErrorCodeToolValue : USINT
GET
                    IF u8ErrorCode.ToolScalingDivisor = 0 OR u8ErrorCode.AppScalingMultiplier = 0 THEN
	_MatchLog^.Error("Get u8ErrorCodeToolValue", "Division by Zero!");
	RETURN;
END_IF

u8ErrorCodeToolValue := TO_USINT(((u8ErrorCode.Value - u8ErrorCode.AppScalingOffset) * u8ErrorCode.AppScalingDivisor / u8ErrorCode.AppScalingMultiplier * u8ErrorCode.ToolScalingMultiplier / u8ErrorCode.ToolScalingDivisor) + u8ErrorCode.ToolScalingOffset);

                  
END_GET
END_PROPERTY

PROPERTY i16DebugVehicleSlopeToolValue : INT
GET
                    IF i16DebugVehicleSlope.ToolScalingDivisor = 0 OR i16DebugVehicleSlope.AppScalingMultiplier = 0 THEN
	_MatchLog^.Error("Get i16DebugVehicleSlopeToolValue", "Division by Zero!");
	RETURN;
END_IF

i16DebugVehicleSlopeToolValue := TO_INT(((i16DebugVehicleSlope.Value - i16DebugVehicleSlope.AppScalingOffset) * i16DebugVehicleSlope.AppScalingDivisor / i16DebugVehicleSlope.AppScalingMultiplier * i16DebugVehicleSlope.ToolScalingMultiplier / i16DebugVehicleSlope.ToolScalingDivisor) + i16DebugVehicleSlope.ToolScalingOffset);

                  
END_GET
END_PROPERTY

METHOD InitializeCanSignals
                  u16FaultyValue.AppScalingDivisor :=1;
u16FaultyValue.AppScalingMultiplier :=1;
u16FaultyValue.AppScalingOffset :=0;
u16FaultyValue.AppUnit :="";
u16FaultyValue.CanDefault :=0;
u16FaultyValue.CanInit :=0;
u16FaultyValue.CanMax :=VBasic.LibConst.U16_MAX;
u16FaultyValue.CanMin :=VBasic.LibConst.U16_MIN;
u16FaultyValue.CanUnit :="";
u16FaultyValue.Description :="new signal";
u16FaultyValue.ErrorReaction := eErrorReaction.ERSIG_DFLT;
u16FaultyValue.ReceiverAdress :=1;
u16FaultyValue.ToolScalingDivisor :=1;
u16FaultyValue.ToolScalingMultiplier :=1;
u16FaultyValue.ToolScalingOffset :=0;
u16FaultyValue.ToolUnit :="";

u8DeviceNum.AppScalingDivisor :=1;
u8DeviceNum.AppScalingMultiplier :=1;
u8DeviceNum.AppScalingOffset :=0;
u8DeviceNum.AppUnit :="";
u8DeviceNum.CanDefault :=0;
u8DeviceNum.CanInit :=0;
u8DeviceNum.CanMax :=VBasic.LibConst.U8_MAX;
u8DeviceNum.CanMin :=VBasic.LibConst.U8_MIN;
u8DeviceNum.CanUnit :="";
u8DeviceNum.Description :="new signal";
u8DeviceNum.ErrorReaction := eErrorReaction.ERSIG_DFLT;
u8DeviceNum.ReceiverAdress :=1;
u8DeviceNum.ToolScalingDivisor :=1;
u8DeviceNum.ToolScalingMultiplier :=1;
u8DeviceNum.ToolScalingOffset :=0;
u8DeviceNum.ToolUnit :="";

u8ErrorCode.AppScalingDivisor :=1;
u8ErrorCode.AppScalingMultiplier :=1;
u8ErrorCode.AppScalingOffset :=0;
u8ErrorCode.AppUnit :="";
u8ErrorCode.CanDefault :=0;
u8ErrorCode.CanInit :=0;
u8ErrorCode.CanMax :=VBasic.LibConst.U8_MAX;
u8ErrorCode.CanMin :=VBasic.LibConst.U8_MIN;
u8ErrorCode.CanUnit :="";
u8ErrorCode.Description :="new signal";
u8ErrorCode.ErrorReaction := eErrorReaction.ERSIG_DFLT;
u8ErrorCode.ReceiverAdress :=1;
u8ErrorCode.ToolScalingDivisor :=1;
u8ErrorCode.ToolScalingMultiplier :=1;
u8ErrorCode.ToolScalingOffset :=0;
u8ErrorCode.ToolUnit :="";

i16DebugVehicleSlope.AppScalingDivisor :=1;
i16DebugVehicleSlope.AppScalingMultiplier :=1;
i16DebugVehicleSlope.AppScalingOffset :=0;
i16DebugVehicleSlope.AppUnit :="";
i16DebugVehicleSlope.CanDefault :=0;
i16DebugVehicleSlope.CanInit :=0;
i16DebugVehicleSlope.CanMax :=32767;
i16DebugVehicleSlope.CanMin :=-32768;
i16DebugVehicleSlope.CanUnit :="";
i16DebugVehicleSlope.Description :="new signal";
i16DebugVehicleSlope.ErrorReaction := eErrorReaction.ERSIG_DFLT;
i16DebugVehicleSlope.ReceiverAdress :=1;
i16DebugVehicleSlope.ToolScalingDivisor :=1;
i16DebugVehicleSlope.ToolScalingMultiplier :=1;
i16DebugVehicleSlope.ToolScalingOffset :=0;
i16DebugVehicleSlope.ToolUnit :="";


                
END_METHOD
END_FUNCTION_BLOCK

FUNCTION_BLOCK Msg1RcvFromEvision7MessageClass EXTENDS CanTransmitMessageClass
  VAR_INPUT
    bogLoginStatus : BoolCanSignalClass;
    bogButtonCalibTurretEncoder : BoolCanSignalClass;
    bogButtonCalibMinMastMeasure : BoolCanSignalClass;
    bogButtonCalibMaxMastMeasure : BoolCanSignalClass;
    boSavePosEncodeurMastButton : BoolCanSignalClass;
    bogActivateMeasuringMast : BoolCanSignalClass;
    boRazDistanceTraveledMastMeasure : BoolCanSignalClass;
    bogOffTrackTestBrakeActivated : BoolCanSignalClass;
    bogOffTrackRunInBrakeActivated : BoolCanSignalClass;
    bogOsciServiceBrakeSelect : BoolCanSignalClass;
    bogFixedServiceBrakeSelect : BoolCanSignalClass;
    bogBothServiceBrakeSelect : BoolCanSignalClass;
    bogOsciParkBrakeSelect : BoolCanSignalClass;
    bogFixedParkBrakeSelect : BoolCanSignalClass;
    bogBothParkBrakeSelect : BoolCanSignalClass;
    bogOsciServiceRunInBrakeSelect : BoolCanSignalClass;
    bogFixedServiceRunInBrakeSelect : BoolCanSignalClass;
    bogBothServiceRunInBrakeSelect : BoolCanSignalClass;
    bogTestBrakePageActive : BoolCanSignalClass;
    bogBreakInBrakePageActive : BoolCanSignalClass;
    bogSerialNumber : BoolCanSignalClass;
    bogBPBasketValidate : BoolCanSignalClass;
    bogKeyFilterOverload : BoolCanSignalClass;
    bogKeyNextMode : BoolCanSignalClass;
    bogKeyPrevMode : BoolCanSignalClass;
    bogKeySignalDanger : BoolCanSignalClass;
    bogKeyFlashLightON : BoolCanSignalClass;
    bogKeyCalibMastMin : BoolCanSignalClass;
    bogKeyCalibMastMax : BoolCanSignalClass;
    bogKeyCalibMastValid : BoolCanSignalClass;
    bogKeyGeneratorActivate : BoolCanSignalClass;
    bogKeyWhiteLights15746 : BoolCanSignalClass;
    bogFixe2ndParkBrakeSelect : BoolCanSignalClass;
    bogOsci2ndParkBrakeSelect : BoolCanSignalClass;
    bogKeyRazController : BoolCanSignalClass;
    Counter : UInt32CanSignalClass;
  END_VAR

            
          

METHOD _sendMessage
                  IF IsValidPointer(fCanManagerPointer,'Msg1RcvFromEvision7') THEN
	fMessage.Clear();
	fMessage.DLC := 8;
	fMessage.SetBool(0, g_CanMessages_Msg1RcvFromEvision7.bogLoginStatus.Value);
	fMessage.SetBool(1, g_CanMessages_Msg1RcvFromEvision7.bogButtonCalibTurretEncoder.Value);
	fMessage.SetBool(2, g_CanMessages_Msg1RcvFromEvision7.bogButtonCalibMinMastMeasure.Value);
	fMessage.SetBool(3, g_CanMessages_Msg1RcvFromEvision7.bogButtonCalibMaxMastMeasure.Value);
	fMessage.SetBool(4, g_CanMessages_Msg1RcvFromEvision7.boSavePosEncodeurMastButton.Value);
	fMessage.SetBool(5, g_CanMessages_Msg1RcvFromEvision7.bogActivateMeasuringMast.Value);
	fMessage.SetBool(6, g_CanMessages_Msg1RcvFromEvision7.boRazDistanceTraveledMastMeasure.Value);
	fMessage.SetBool(7, g_CanMessages_Msg1RcvFromEvision7.bogOffTrackTestBrakeActivated.Value);
	fMessage.SetBool(8, g_CanMessages_Msg1RcvFromEvision7.bogOffTrackRunInBrakeActivated.Value);
	fMessage.SetBool(9, g_CanMessages_Msg1RcvFromEvision7.bogOsciServiceBrakeSelect.Value);
	fMessage.SetBool(10, g_CanMessages_Msg1RcvFromEvision7.bogFixedServiceBrakeSelect.Value);
	fMessage.SetBool(11, g_CanMessages_Msg1RcvFromEvision7.bogBothServiceBrakeSelect.Value);
	fMessage.SetBool(12, g_CanMessages_Msg1RcvFromEvision7.bogOsciParkBrakeSelect.Value);
	fMessage.SetBool(13, g_CanMessages_Msg1RcvFromEvision7.bogFixedParkBrakeSelect.Value);
	fMessage.SetBool(14, g_CanMessages_Msg1RcvFromEvision7.bogBothParkBrakeSelect.Value);
	fMessage.SetBool(15, g_CanMessages_Msg1RcvFromEvision7.bogOsciServiceRunInBrakeSelect.Value);
	fMessage.SetBool(16, g_CanMessages_Msg1RcvFromEvision7.bogFixedServiceRunInBrakeSelect.Value);
	fMessage.SetBool(17, g_CanMessages_Msg1RcvFromEvision7.bogBothServiceRunInBrakeSelect.Value);
	fMessage.SetBool(18, g_CanMessages_Msg1RcvFromEvision7.bogTestBrakePageActive.Value);
	fMessage.SetBool(19, g_CanMessages_Msg1RcvFromEvision7.bogBreakInBrakePageActive.Value);
	fMessage.SetBool(20, g_CanMessages_Msg1RcvFromEvision7.bogSerialNumber.Value);
	fMessage.SetBool(21, g_CanMessages_Msg1RcvFromEvision7.bogBPBasketValidate.Value);
	fMessage.SetBool(22, g_CanMessages_Msg1RcvFromEvision7.bogKeyFilterOverload.Value);
	fMessage.SetBool(23, g_CanMessages_Msg1RcvFromEvision7.bogKeyNextMode.Value);
	fMessage.SetBool(24, g_CanMessages_Msg1RcvFromEvision7.bogKeyPrevMode.Value);
	fMessage.SetBool(25, g_CanMessages_Msg1RcvFromEvision7.bogKeySignalDanger.Value);
	fMessage.SetBool(26, g_CanMessages_Msg1RcvFromEvision7.bogKeyFlashLightON.Value);
	fMessage.SetBool(27, g_CanMessages_Msg1RcvFromEvision7.bogKeyCalibMastMin.Value);
	fMessage.SetBool(28, g_CanMessages_Msg1RcvFromEvision7.bogKeyCalibMastMax.Value);
	fMessage.SetBool(29, g_CanMessages_Msg1RcvFromEvision7.bogKeyCalibMastValid.Value);
	fMessage.SetBool(30, g_CanMessages_Msg1RcvFromEvision7.bogKeyGeneratorActivate.Value);
	fMessage.SetBool(31, g_CanMessages_Msg1RcvFromEvision7.bogKeyWhiteLights15746.Value);
	fMessage.SetBool(32, g_CanMessages_Msg1RcvFromEvision7.bogFixe2ndParkBrakeSelect.Value);
	fMessage.SetBool(33, g_CanMessages_Msg1RcvFromEvision7.bogOsci2ndParkBrakeSelect.Value);
	fMessage.SetBool(34, g_CanMessages_Msg1RcvFromEvision7.bogKeyRazController.Value);
	fCanManagerPointer^.SendMessageImmediately(ADR(fMessage),FALSE);
	Counter.Value := Counter.Value + 1;
	fDataChanged := FALSE;
END_IF

                
END_METHOD

PROPERTY bogLoginStatusRawValue : BOOL
GET
                    bogLoginStatusRawValue := bogLoginStatus.Value;

                  
END_GET
SET
                    bogLoginStatus.Value := bogLoginStatusRawValue;

                  
END_SET
END_PROPERTY

PROPERTY bogButtonCalibTurretEncoderRawValue : BOOL
GET
                    bogButtonCalibTurretEncoderRawValue := bogButtonCalibTurretEncoder.Value;

                  
END_GET
SET
                    bogButtonCalibTurretEncoder.Value := bogButtonCalibTurretEncoderRawValue;

                  
END_SET
END_PROPERTY

PROPERTY bogButtonCalibMinMastMeasureRawValue : BOOL
GET
                    bogButtonCalibMinMastMeasureRawValue := bogButtonCalibMinMastMeasure.Value;

                  
END_GET
SET
                    bogButtonCalibMinMastMeasure.Value := bogButtonCalibMinMastMeasureRawValue;

                  
END_SET
END_PROPERTY

PROPERTY bogButtonCalibMaxMastMeasureRawValue : BOOL
GET
                    bogButtonCalibMaxMastMeasureRawValue := bogButtonCalibMaxMastMeasure.Value;

                  
END_GET
SET
                    bogButtonCalibMaxMastMeasure.Value := bogButtonCalibMaxMastMeasureRawValue;

                  
END_SET
END_PROPERTY

PROPERTY boSavePosEncodeurMastButtonRawValue : BOOL
GET
                    boSavePosEncodeurMastButtonRawValue := boSavePosEncodeurMastButton.Value;

                  
END_GET
SET
                    boSavePosEncodeurMastButton.Value := boSavePosEncodeurMastButtonRawValue;

                  
END_SET
END_PROPERTY

PROPERTY bogActivateMeasuringMastRawValue : BOOL
GET
                    bogActivateMeasuringMastRawValue := bogActivateMeasuringMast.Value;

                  
END_GET
SET
                    bogActivateMeasuringMast.Value := bogActivateMeasuringMastRawValue;

                  
END_SET
END_PROPERTY

PROPERTY boRazDistanceTraveledMastMeasureRawValue : BOOL
GET
                    boRazDistanceTraveledMastMeasureRawValue := boRazDistanceTraveledMastMeasure.Value;

                  
END_GET
SET
                    boRazDistanceTraveledMastMeasure.Value := boRazDistanceTraveledMastMeasureRawValue;

                  
END_SET
END_PROPERTY

PROPERTY bogOffTrackTestBrakeActivatedRawValue : BOOL
GET
                    bogOffTrackTestBrakeActivatedRawValue := bogOffTrackTestBrakeActivated.Value;

                  
END_GET
SET
                    bogOffTrackTestBrakeActivated.Value := bogOffTrackTestBrakeActivatedRawValue;

                  
END_SET
END_PROPERTY

PROPERTY bogOffTrackRunInBrakeActivatedRawValue : BOOL
GET
                    bogOffTrackRunInBrakeActivatedRawValue := bogOffTrackRunInBrakeActivated.Value;

                  
END_GET
SET
                    bogOffTrackRunInBrakeActivated.Value := bogOffTrackRunInBrakeActivatedRawValue;

                  
END_SET
END_PROPERTY

PROPERTY bogOsciServiceBrakeSelectRawValue : BOOL
GET
                    bogOsciServiceBrakeSelectRawValue := bogOsciServiceBrakeSelect.Value;

                  
END_GET
SET
                    bogOsciServiceBrakeSelect.Value := bogOsciServiceBrakeSelectRawValue;

                  
END_SET
END_PROPERTY

PROPERTY bogFixedServiceBrakeSelectRawValue : BOOL
GET
                    bogFixedServiceBrakeSelectRawValue := bogFixedServiceBrakeSelect.Value;

                  
END_GET
SET
                    bogFixedServiceBrakeSelect.Value := bogFixedServiceBrakeSelectRawValue;

                  
END_SET
END_PROPERTY

PROPERTY bogBothServiceBrakeSelectRawValue : BOOL
GET
                    bogBothServiceBrakeSelectRawValue := bogBothServiceBrakeSelect.Value;

                  
END_GET
SET
                    bogBothServiceBrakeSelect.Value := bogBothServiceBrakeSelectRawValue;

                  
END_SET
END_PROPERTY

PROPERTY bogOsciParkBrakeSelectRawValue : BOOL
GET
                    bogOsciParkBrakeSelectRawValue := bogOsciParkBrakeSelect.Value;

                  
END_GET
SET
                    bogOsciParkBrakeSelect.Value := bogOsciParkBrakeSelectRawValue;

                  
END_SET
END_PROPERTY

PROPERTY bogFixedParkBrakeSelectRawValue : BOOL
GET
                    bogFixedParkBrakeSelectRawValue := bogFixedParkBrakeSelect.Value;

                  
END_GET
SET
                    bogFixedParkBrakeSelect.Value := bogFixedParkBrakeSelectRawValue;

                  
END_SET
END_PROPERTY

PROPERTY bogBothParkBrakeSelectRawValue : BOOL
GET
                    bogBothParkBrakeSelectRawValue := bogBothParkBrakeSelect.Value;

                  
END_GET
SET
                    bogBothParkBrakeSelect.Value := bogBothParkBrakeSelectRawValue;

                  
END_SET
END_PROPERTY

PROPERTY bogOsciServiceRunInBrakeSelectRawValue : BOOL
GET
                    bogOsciServiceRunInBrakeSelectRawValue := bogOsciServiceRunInBrakeSelect.Value;

                  
END_GET
SET
                    bogOsciServiceRunInBrakeSelect.Value := bogOsciServiceRunInBrakeSelectRawValue;

                  
END_SET
END_PROPERTY

PROPERTY bogFixedServiceRunInBrakeSelectRawValue : BOOL
GET
                    bogFixedServiceRunInBrakeSelectRawValue := bogFixedServiceRunInBrakeSelect.Value;

                  
END_GET
SET
                    bogFixedServiceRunInBrakeSelect.Value := bogFixedServiceRunInBrakeSelectRawValue;

                  
END_SET
END_PROPERTY

PROPERTY bogBothServiceRunInBrakeSelectRawValue : BOOL
GET
                    bogBothServiceRunInBrakeSelectRawValue := bogBothServiceRunInBrakeSelect.Value;

                  
END_GET
SET
                    bogBothServiceRunInBrakeSelect.Value := bogBothServiceRunInBrakeSelectRawValue;

                  
END_SET
END_PROPERTY

PROPERTY bogTestBrakePageActiveRawValue : BOOL
GET
                    bogTestBrakePageActiveRawValue := bogTestBrakePageActive.Value;

                  
END_GET
SET
                    bogTestBrakePageActive.Value := bogTestBrakePageActiveRawValue;

                  
END_SET
END_PROPERTY

PROPERTY bogBreakInBrakePageActiveRawValue : BOOL
GET
                    bogBreakInBrakePageActiveRawValue := bogBreakInBrakePageActive.Value;

                  
END_GET
SET
                    bogBreakInBrakePageActive.Value := bogBreakInBrakePageActiveRawValue;

                  
END_SET
END_PROPERTY

PROPERTY bogSerialNumberRawValue : BOOL
GET
                    bogSerialNumberRawValue := bogSerialNumber.Value;

                  
END_GET
SET
                    bogSerialNumber.Value := bogSerialNumberRawValue;

                  
END_SET
END_PROPERTY

PROPERTY bogBPBasketValidateRawValue : BOOL
GET
                    bogBPBasketValidateRawValue := bogBPBasketValidate.Value;

                  
END_GET
SET
                    bogBPBasketValidate.Value := bogBPBasketValidateRawValue;

                  
END_SET
END_PROPERTY

PROPERTY bogKeyFilterOverloadRawValue : BOOL
GET
                    bogKeyFilterOverloadRawValue := bogKeyFilterOverload.Value;

                  
END_GET
SET
                    bogKeyFilterOverload.Value := bogKeyFilterOverloadRawValue;

                  
END_SET
END_PROPERTY

PROPERTY bogKeyNextModeRawValue : BOOL
GET
                    bogKeyNextModeRawValue := bogKeyNextMode.Value;

                  
END_GET
SET
                    bogKeyNextMode.Value := bogKeyNextModeRawValue;

                  
END_SET
END_PROPERTY

PROPERTY bogKeyPrevModeRawValue : BOOL
GET
                    bogKeyPrevModeRawValue := bogKeyPrevMode.Value;

                  
END_GET
SET
                    bogKeyPrevMode.Value := bogKeyPrevModeRawValue;

                  
END_SET
END_PROPERTY

PROPERTY bogKeySignalDangerRawValue : BOOL
GET
                    bogKeySignalDangerRawValue := bogKeySignalDanger.Value;

                  
END_GET
SET
                    bogKeySignalDanger.Value := bogKeySignalDangerRawValue;

                  
END_SET
END_PROPERTY

PROPERTY bogKeyFlashLightONRawValue : BOOL
GET
                    bogKeyFlashLightONRawValue := bogKeyFlashLightON.Value;

                  
END_GET
SET
                    bogKeyFlashLightON.Value := bogKeyFlashLightONRawValue;

                  
END_SET
END_PROPERTY

PROPERTY bogKeyCalibMastMinRawValue : BOOL
GET
                    bogKeyCalibMastMinRawValue := bogKeyCalibMastMin.Value;

                  
END_GET
SET
                    bogKeyCalibMastMin.Value := bogKeyCalibMastMinRawValue;

                  
END_SET
END_PROPERTY

PROPERTY bogKeyCalibMastMaxRawValue : BOOL
GET
                    bogKeyCalibMastMaxRawValue := bogKeyCalibMastMax.Value;

                  
END_GET
SET
                    bogKeyCalibMastMax.Value := bogKeyCalibMastMaxRawValue;

                  
END_SET
END_PROPERTY

PROPERTY bogKeyCalibMastValidRawValue : BOOL
GET
                    bogKeyCalibMastValidRawValue := bogKeyCalibMastValid.Value;

                  
END_GET
SET
                    bogKeyCalibMastValid.Value := bogKeyCalibMastValidRawValue;

                  
END_SET
END_PROPERTY

PROPERTY bogKeyGeneratorActivateRawValue : BOOL
GET
                    bogKeyGeneratorActivateRawValue := bogKeyGeneratorActivate.Value;

                  
END_GET
SET
                    bogKeyGeneratorActivate.Value := bogKeyGeneratorActivateRawValue;

                  
END_SET
END_PROPERTY

PROPERTY bogKeyWhiteLights15746RawValue : BOOL
GET
                    bogKeyWhiteLights15746RawValue := bogKeyWhiteLights15746.Value;

                  
END_GET
SET
                    bogKeyWhiteLights15746.Value := bogKeyWhiteLights15746RawValue;

                  
END_SET
END_PROPERTY

PROPERTY bogFixe2ndParkBrakeSelectRawValue : BOOL
GET
                    bogFixe2ndParkBrakeSelectRawValue := bogFixe2ndParkBrakeSelect.Value;

                  
END_GET
SET
                    bogFixe2ndParkBrakeSelect.Value := bogFixe2ndParkBrakeSelectRawValue;

                  
END_SET
END_PROPERTY

PROPERTY bogOsci2ndParkBrakeSelectRawValue : BOOL
GET
                    bogOsci2ndParkBrakeSelectRawValue := bogOsci2ndParkBrakeSelect.Value;

                  
END_GET
SET
                    bogOsci2ndParkBrakeSelect.Value := bogOsci2ndParkBrakeSelectRawValue;

                  
END_SET
END_PROPERTY

PROPERTY bogKeyRazControllerRawValue : BOOL
GET
                    bogKeyRazControllerRawValue := bogKeyRazController.Value;

                  
END_GET
SET
                    bogKeyRazController.Value := bogKeyRazControllerRawValue;

                  
END_SET
END_PROPERTY

PROPERTY bogLoginStatusToolValue : BOOL
GET
                    bogLoginStatusToolValue := bogLoginStatus.Value;

                  
END_GET
SET
                    bogLoginStatus.Value := bogLoginStatusToolValue;

                  
END_SET
END_PROPERTY

PROPERTY bogButtonCalibTurretEncoderToolValue : BOOL
GET
                    bogButtonCalibTurretEncoderToolValue := bogButtonCalibTurretEncoder.Value;

                  
END_GET
SET
                    bogButtonCalibTurretEncoder.Value := bogButtonCalibTurretEncoderToolValue;

                  
END_SET
END_PROPERTY

PROPERTY bogButtonCalibMinMastMeasureToolValue : BOOL
GET
                    bogButtonCalibMinMastMeasureToolValue := bogButtonCalibMinMastMeasure.Value;

                  
END_GET
SET
                    bogButtonCalibMinMastMeasure.Value := bogButtonCalibMinMastMeasureToolValue;

                  
END_SET
END_PROPERTY

PROPERTY bogButtonCalibMaxMastMeasureToolValue : BOOL
GET
                    bogButtonCalibMaxMastMeasureToolValue := bogButtonCalibMaxMastMeasure.Value;

                  
END_GET
SET
                    bogButtonCalibMaxMastMeasure.Value := bogButtonCalibMaxMastMeasureToolValue;

                  
END_SET
END_PROPERTY

PROPERTY boSavePosEncodeurMastButtonToolValue : BOOL
GET
                    boSavePosEncodeurMastButtonToolValue := boSavePosEncodeurMastButton.Value;

                  
END_GET
SET
                    boSavePosEncodeurMastButton.Value := boSavePosEncodeurMastButtonToolValue;

                  
END_SET
END_PROPERTY

PROPERTY bogActivateMeasuringMastToolValue : BOOL
GET
                    bogActivateMeasuringMastToolValue := bogActivateMeasuringMast.Value;

                  
END_GET
SET
                    bogActivateMeasuringMast.Value := bogActivateMeasuringMastToolValue;

                  
END_SET
END_PROPERTY

PROPERTY boRazDistanceTraveledMastMeasureToolValue : BOOL
GET
                    boRazDistanceTraveledMastMeasureToolValue := boRazDistanceTraveledMastMeasure.Value;

                  
END_GET
SET
                    boRazDistanceTraveledMastMeasure.Value := boRazDistanceTraveledMastMeasureToolValue;

                  
END_SET
END_PROPERTY

PROPERTY bogOffTrackTestBrakeActivatedToolValue : BOOL
GET
                    bogOffTrackTestBrakeActivatedToolValue := bogOffTrackTestBrakeActivated.Value;

                  
END_GET
SET
                    bogOffTrackTestBrakeActivated.Value := bogOffTrackTestBrakeActivatedToolValue;

                  
END_SET
END_PROPERTY

PROPERTY bogOffTrackRunInBrakeActivatedToolValue : BOOL
GET
                    bogOffTrackRunInBrakeActivatedToolValue := bogOffTrackRunInBrakeActivated.Value;

                  
END_GET
SET
                    bogOffTrackRunInBrakeActivated.Value := bogOffTrackRunInBrakeActivatedToolValue;

                  
END_SET
END_PROPERTY

PROPERTY bogOsciServiceBrakeSelectToolValue : BOOL
GET
                    bogOsciServiceBrakeSelectToolValue := bogOsciServiceBrakeSelect.Value;

                  
END_GET
SET
                    bogOsciServiceBrakeSelect.Value := bogOsciServiceBrakeSelectToolValue;

                  
END_SET
END_PROPERTY

PROPERTY bogFixedServiceBrakeSelectToolValue : BOOL
GET
                    bogFixedServiceBrakeSelectToolValue := bogFixedServiceBrakeSelect.Value;

                  
END_GET
SET
                    bogFixedServiceBrakeSelect.Value := bogFixedServiceBrakeSelectToolValue;

                  
END_SET
END_PROPERTY

PROPERTY bogBothServiceBrakeSelectToolValue : BOOL
GET
                    bogBothServiceBrakeSelectToolValue := bogBothServiceBrakeSelect.Value;

                  
END_GET
SET
                    bogBothServiceBrakeSelect.Value := bogBothServiceBrakeSelectToolValue;

                  
END_SET
END_PROPERTY

PROPERTY bogOsciParkBrakeSelectToolValue : BOOL
GET
                    bogOsciParkBrakeSelectToolValue := bogOsciParkBrakeSelect.Value;

                  
END_GET
SET
                    bogOsciParkBrakeSelect.Value := bogOsciParkBrakeSelectToolValue;

                  
END_SET
END_PROPERTY

PROPERTY bogFixedParkBrakeSelectToolValue : BOOL
GET
                    bogFixedParkBrakeSelectToolValue := bogFixedParkBrakeSelect.Value;

                  
END_GET
SET
                    bogFixedParkBrakeSelect.Value := bogFixedParkBrakeSelectToolValue;

                  
END_SET
END_PROPERTY

PROPERTY bogBothParkBrakeSelectToolValue : BOOL
GET
                    bogBothParkBrakeSelectToolValue := bogBothParkBrakeSelect.Value;

                  
END_GET
SET
                    bogBothParkBrakeSelect.Value := bogBothParkBrakeSelectToolValue;

                  
END_SET
END_PROPERTY

PROPERTY bogOsciServiceRunInBrakeSelectToolValue : BOOL
GET
                    bogOsciServiceRunInBrakeSelectToolValue := bogOsciServiceRunInBrakeSelect.Value;

                  
END_GET
SET
                    bogOsciServiceRunInBrakeSelect.Value := bogOsciServiceRunInBrakeSelectToolValue;

                  
END_SET
END_PROPERTY

PROPERTY bogFixedServiceRunInBrakeSelectToolValue : BOOL
GET
                    bogFixedServiceRunInBrakeSelectToolValue := bogFixedServiceRunInBrakeSelect.Value;

                  
END_GET
SET
                    bogFixedServiceRunInBrakeSelect.Value := bogFixedServiceRunInBrakeSelectToolValue;

                  
END_SET
END_PROPERTY

PROPERTY bogBothServiceRunInBrakeSelectToolValue : BOOL
GET
                    bogBothServiceRunInBrakeSelectToolValue := bogBothServiceRunInBrakeSelect.Value;

                  
END_GET
SET
                    bogBothServiceRunInBrakeSelect.Value := bogBothServiceRunInBrakeSelectToolValue;

                  
END_SET
END_PROPERTY

PROPERTY bogTestBrakePageActiveToolValue : BOOL
GET
                    bogTestBrakePageActiveToolValue := bogTestBrakePageActive.Value;

                  
END_GET
SET
                    bogTestBrakePageActive.Value := bogTestBrakePageActiveToolValue;

                  
END_SET
END_PROPERTY

PROPERTY bogBreakInBrakePageActiveToolValue : BOOL
GET
                    bogBreakInBrakePageActiveToolValue := bogBreakInBrakePageActive.Value;

                  
END_GET
SET
                    bogBreakInBrakePageActive.Value := bogBreakInBrakePageActiveToolValue;

                  
END_SET
END_PROPERTY

PROPERTY bogSerialNumberToolValue : BOOL
GET
                    bogSerialNumberToolValue := bogSerialNumber.Value;

                  
END_GET
SET
                    bogSerialNumber.Value := bogSerialNumberToolValue;

                  
END_SET
END_PROPERTY

PROPERTY bogBPBasketValidateToolValue : BOOL
GET
                    bogBPBasketValidateToolValue := bogBPBasketValidate.Value;

                  
END_GET
SET
                    bogBPBasketValidate.Value := bogBPBasketValidateToolValue;

                  
END_SET
END_PROPERTY

